ABB RAPID module: Module1.mod

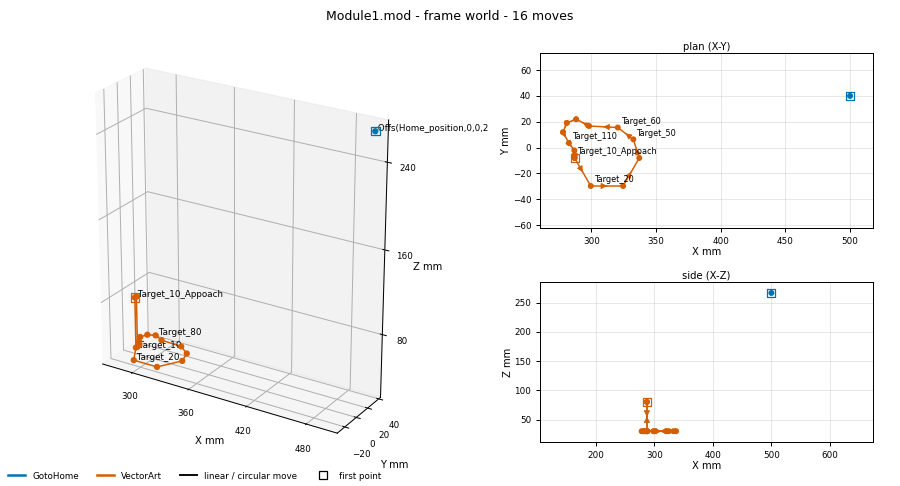
[picture p0: tool path of Module1.mod in frame world, 16 of 848 moves have a stored position in this frame; points joined in program order, loops and branches not executed]
MODULE Module1
    ! Define Global Constants
	CONST robtarget Home_position:=[[297,210,180],[0,0,1,0],[0,0,0,0],[9E+09,9E+09,9E+09,9E+09,9E+09,9E+09]];
	CONST robtarget Bottom_Left:=[[0,420,0],[0,0,1,0],[0,0,0,0],[9E+09,9E+09,9E+09,9E+09,9E+09,9E+09]];
	CONST robtarget Top_Left:=[[297,420,0],[0,0,1,0],[0,0,0,0],[9E+09,9E+09,9E+09,9E+09,9E+09,9E+09]];
	CONST robtarget Top_Right:=[[297,0,0],[0,0,1,0],[0,0,0,0],[9E+09,9E+09,9E+09,9E+09,9E+09,9E+09]];
	CONST robtarget Bottom_Right:=[[0,0,0],[0,0,1,0],[0,0,0,0],[9E+09,9E+09,9E+09,9E+09,9E+09,9E+09]];
	CONST robtarget Target_10_Appoach:=[[84,162,13.48],[0,-0.707106781,0.707106781,0],[-1,0,-2,0],[9E+09,9E+09,9E+09,9E+09,9E+09,9E+09]];
	CONST robtarget Target_10:=[[84,162,-36.52],[0,-0.707106781,0.707106781,0],[-1,0,-2,0],[9E+09,9E+09,9E+09,9E+09,9E+09,9E+09]];
	CONST robtarget Target_20:=[[96.5,140.349364905,-36.52],[0,-0.707106781,0.707106781,0],[-1,0,-2,0],[9E+09,9E+09,9E+09,9E+09,9E+09,9E+09]];
	CONST robtarget Target_30:=[[121.5,140.349364905,-36.52],[0,-0.707106781,0.707106781,0],[-1,0,-2,0],[9E+09,9E+09,9E+09,9E+09,9E+09,9E+09]];
	CONST robtarget Target_40:=[[134,162,-36.52],[0,-0.707106781,0.707106781,0],[-1,0,-2,0],[9E+09,9E+09,9E+09,9E+09,9E+09,9E+09]];
	CONST robtarget Target_50:=[[129.425575437,176.415126364,-36.52],[0,-0.707106781,0.707106781,0],[0,0,-1,0],[9E+09,9E+09,9E+09,9E+09,9E+09,9E+09]];
	CONST robtarget Target_60:=[[117.376330553,185.554980078,-36.52],[0,-0.707106781,0.707106781,0],[0,0,-1,0],[9E+09,9E+09,9E+09,9E+09,9E+09,9E+09]];
	CONST robtarget Target_70:=[[95.190280659,186.713087817,-36.52],[0,-0.707106781,0.707106781,0],[0,0,-1,0],[9E+09,9E+09,9E+09,9E+09,9E+09,9E+09]];
	CONST robtarget Target_80:=[[85.203125494,191.997936789,-36.52],[0,-0.707106781,0.707106781,0],[0,0,-1,0],[9E+09,9E+09,9E+09,9E+09,9E+09,9E+09]];
	CONST robtarget Target_90:=[[78.001116337,189.142522487,-36.52],[0,-0.707106781,0.707106781,0],[0,0,-1,0],[9E+09,9E+09,9E+09,9E+09,9E+09,9E+09]];
	CONST robtarget Target_100:=[[75,182,-36.52],[0,-0.707106781,0.707106781,0],[0,0,-1,0],[9E+09,9E+09,9E+09,9E+09,9E+09,9E+09]];
	CONST robtarget Target_110:=[[79.573343373,173.600512048,-36.52],[0,-0.707106781,0.707106781,0],[0,0,-1,0],[9E+09,9E+09,9E+09,9E+09,9E+09,9E+09]];
	CONST robtarget Target_120:=[[83.780815333,167.881241697,-36.52],[0,-0.707106781,0.707106781,0],[-1,0,-2,0],[9E+09,9E+09,9E+09,9E+09,9E+09,9E+09]];
	CONST robtarget Target_130:=[[84.104776248,164.286445783,-36.52],[0,-0.707106781,0.707106781,0],[-1,0,-2,0],[9E+09,9E+09,9E+09,9E+09,9E+09,9E+09]];
	CONST robtarget Target_130_Depart:=[[84.104776248,164.286445783,13.48],[0,-0.707106781,0.707106781,0],[-1,0,-2,0],[9E+09,9E+09,9E+09,9E+09,9E+09,9E+09]];

    !***********************************************************
    !
    ! Module:  Module1
    !
    ! Disclaimer:
    !    This module was written as part of my submission for Middlesex University's
    !    2017-2018 Mobile Robots and Manipulators module.
    !
    !    Note that this script in intended for GOOD and not for EVIL.
    !    Please do not use in any negative context, at least not without prior consent from
    !    the author of this script.
    !
    ! Author:
    !    Chibuike Okpaluba <co607@live.mdx.ac.uk> M00543047
    !
    ! Module Tutor:
    !    Dr Aleksander Zivanovic <a.zivanovic@mdx.ac.uk>
    !
    ! Description:
    !   This module contains all the necessary procedures and functions required to
    !
    !   1. Draw manually defined characters on a given worksurface using a preselected tool.
    !   2. Draw selected artworks on a given worksurface using a preselected tool.
    !   3. Draw the vector artwork on a given worksurface using a preselected tool.
    !   4. Automatically generate artworks for users that select the special option.
    !
    !   -- THE ENTRY POINT FOR THIS MODULE IS MAIN --
    !
    ! Version:
    !   v1.0
    !
    ! Questions and Answers:
    !   For more information please email the author of the module
    !
    !
    ! Thank you.
    !
    !***********************************************************


    !***********************************************************
    !
    ! Procedure main
    !   This the entry point of this module.
    !
    !   This procedure executes other procedures based on user inputs
    !***********************************************************
    PROC Main()
        ! Define Function Variables
        VAR num font_size := 0.5;
        VAR string answer := "Blink";

        ! GO Home and Wait 10 seconds
        GotoHome;
        !WaitTime 10;

        ! Get Data from the user
        TPReadFK reg1, "Select Drawing?", "Initials", "Artwork", "Vector", "Your String", "Special";

        ! Execute based on user data
        IF reg1 = 1 THEN
            TPWrite "Drawing initials: ''C.O''";
            DrawIntials font_size;

        ELSEIF reg1 = 2 THEN
            TPWrite "Drawing Artwork";
            DrawArtwork v100, v50, 100, 25, -10, 50;

        ELSEIF reg1 = 3 THEN
            TPWrite "Drawing Vector Art";
            VectorArt;

        ELSEIF reg1 = 4 THEN
            ! Get Text from the user
            answer := UIAlphaEntry(\Header:="Blink UI",
                \Message:="Enter your text?"
                \Icon:=iconInfo
                \InitString:="Your Text");

            ! Get font size from the user
            TPReadNum reg1, "Enter your font_size";

            ! Draw the users string
            DrawString answer, reg1, v80, v50, 10, 10, -10, 50;

        ELSEIF reg1 = 5 THEN
            ! Start special art
            MakeArtwork;

        ELSE
            TPWrite "Invalid selection";

        ENDIF

    ENDPROC

    !***********************************************************
    !
    ! Procedure GotoHome
    !   This Procedure moves the arm to the GLOBAL defined home position
    !
    ! Example
    !   GotoHome
    !
    !***********************************************************
    PROC GotoHome()
        ! Move arm joints to home position
        MoveJ Offs(Home_position, 0, 0, 20),v1000,z100,tool0\WObj:=WorkSurface;
    ENDPROC

    !***********************************************************
    !
    ! Procedure DrawIntials
    !   This procedure draws the intials on the work surface
    !
    ! Example
    !   VAR num font_size := 1.0;
    !   DrawIntials font_size;
    !
    !***********************************************************
    PROC DrawIntials(num font_size)
        DrawString "#Chib!", font_size, v100, v50, 5, 5, -10, 50;
        DrawString "#Chib!", font_size, v100, v50, 5, 65, -10, 50;
        DrawString "#Chib!", font_size, v100, v50, 5, 125, -10, 50;
        DrawString "#Chib!", font_size, v100, v50, 5, 185, -10, 50;
    ENDPROC

    !***********************************************************
    !
    ! Procedure MakeArtwork
    !   This procedure creates an artwork for the user based on the users string input
    !
    ! Example
    !   MakeArtwork;
    !
    !***********************************************************
    PROC MakeArtwork()
        VAR num page_width := 290;
        VAR num x_padding := 55;
        VAR num y_padding := 50;
        VAR string input_string := "";
        VAR num font_size := 0;

        VAR num z_offset := -10;
        VAR num penup_offset := 50;

        VAR num art_option;

        ! Get User's text
        input_string := UIAlphaEntry(\Header:="Blink UI",
                \Message:="Enter your text?"
                \Icon:=iconInfo
                \InitString:="#YourText");

        ! Drawing border art
        DrawArtWork_ArtBorder 0.45, v100, v50, 0, 0, z_offset, penup_offset;

        ! Calculate ideal font size
        font_size := get_ideal_font_size(input_string, page_width, x_padding);

        y_padding := 200 - (font_size * 50);
        DrawString input_string, font_size, v100, v50, x_padding, y_padding, z_offset, penup_offset;

        ! Get art option from the user
        TPReadFK reg1, "Select Art Option?", "House", stEmpty, stEmpty, stEmpty, "Glasses";
        art_option := reg1;

        IF art_option = 5 THEN
            y_padding := y_padding + (50 * font_size) + 5;
            x_padding := 96;
            DrawArtWork_Glasses 0.47, v100, v50, x_padding, y_padding, z_offset, penup_offset;
        ELSEIF art_option = 1 THEN
            y_padding := y_padding + (50 * font_size) + 5;
            x_padding := 106;
            DrawArtWork_House 0.38, v100, v50, x_padding, y_padding, z_offset, penup_offset;
        ENDIF
    ENDPROC

    !***********************************************************
    !
    ! Procedure DrawArtwork
    !   This procedure draws my artwork on the work surface
    !
    ! Example
    !   VAR speeddata approach_speed := v100;  // Approach speed for arm
    !   VAR speeddata write_speed := v80;      // Write speed for arm
    !   VAR num x_offset := 0;                 // x offset from worksurface origin
    !   VAR num y_offset := 0;                 // y offset from worksurface origin
    !   VAR num z_offset := 0;                 // z offset from worksurface origin
    !   VAR num pen_offset := 30;              // Defines pen position for pen up
    !
    !   DrawArtwork approach_speed, write_speed, x_offset, y_offset, z_offset, penup_offset;
    !
    !***********************************************************
    PROC DrawArtwork(speeddata approach_speed, speeddata write_speed, num x_offset, num y_offset, num z_offset, num penup_offset)
        ! Define all points for artwork
        VAR pos pos0{17} := [[153.29999999999998, 151.89999999999998, 0],[152.6, 152.6, 0],[152.6, 154.0, 0],[153.29999999999998, 154.7, 0],[153.29999999999998, 155.39999999999998, 0],[155.39999999999998, 157.5, 0],[158.2, 157.5, 0],[160.29999999999998, 155.39999999999998, 0],[160.29999999999998, 154.7, 0],[161.0, 154.0, 0],[161.0, 152.6, 0],[160.29999999999998, 151.89999999999998, 0],[160.29999999999998, 151.2, 0],[158.89999999999998, 149.79999999999998, 0],[154.7, 149.79999999999998, 0],[153.29999999999998, 151.2, 0],[153.29999999999998, 151.89999999999998, 0]];
        VAR pos pos1{10} := [[154.7, 152.6, 0],[155.39999999999998, 151.89999999999998, 0],[156.79999999999998, 151.89999999999998, 0],[157.5, 152.6, 0],[157.5, 154.0, 0],[156.79999999999998, 154.0, 0],[156.1, 154.7, 0],[155.39999999999998, 154.0, 0],[154.7, 154.0, 0],[154.7, 152.6, 0]];
        VAR pos pos2{17} := [[153.29999999999998, 109.19999999999999, 0],[152.6, 109.89999999999999, 0],[152.6, 111.3, 0],[153.29999999999998, 112.0, 0],[153.29999999999998, 112.69999999999999, 0],[155.39999999999998, 114.8, 0],[158.2, 114.8, 0],[160.29999999999998, 112.69999999999999, 0],[160.29999999999998, 112.0, 0],[161.0, 111.3, 0],[161.0, 109.89999999999999, 0],[160.29999999999998, 109.19999999999999, 0],[160.29999999999998, 108.5, 0],[158.89999999999998, 107.1, 0],[154.7, 107.1, 0],[153.29999999999998, 108.5, 0],[153.29999999999998, 109.19999999999999, 0]];
        VAR pos pos3{10} := [[154.7, 109.89999999999999, 0],[155.39999999999998, 109.19999999999999, 0],[156.79999999999998, 109.19999999999999, 0],[157.5, 109.89999999999999, 0],[157.5, 111.3, 0],[156.79999999999998, 111.3, 0],[156.1, 112.0, 0],[155.39999999999998, 111.3, 0],[154.7, 111.3, 0],[154.7, 109.89999999999999, 0]];
        VAR pos pos4{19} := [[153.29999999999998, 82.6, 0],[152.6, 83.3, 0],[152.6, 84.69999999999999, 0],[153.29999999999998, 85.39999999999999, 0],[153.29999999999998, 86.1, 0],[155.39999999999998, 88.19999999999999, 0],[158.2, 88.19999999999999, 0],[160.29999999999998, 86.1, 0],[160.29999999999998, 85.39999999999999, 0],[161.0, 84.69999999999999, 0],[161.0, 83.3, 0],[160.29999999999998, 82.6, 0],[160.29999999999998, 81.89999999999999, 0],[159.6, 81.19999999999999, 0],[158.89999999999998, 81.19999999999999, 0],[158.2, 80.5, 0],[154.7, 80.5, 0],[153.29999999999998, 81.89999999999999, 0],[153.29999999999998, 82.6, 0]];
        VAR pos pos5{10} := [[154.7, 83.3, 0],[155.39999999999998, 82.6, 0],[156.79999999999998, 82.6, 0],[157.5, 83.3, 0],[157.5, 84.69999999999999, 0],[156.79999999999998, 84.69999999999999, 0],[156.1, 85.39999999999999, 0],[155.39999999999998, 84.69999999999999, 0],[154.7, 84.69999999999999, 0],[154.7, 83.3, 0]];
        VAR pos pos6{57} := [[126.69999999999999, 172.89999999999998, 0],[125.99999999999999, 173.6, 0],[125.99999999999999, 177.79999999999998, 0],[126.69999999999999, 178.5, 0],[126.69999999999999, 180.6, 0],[127.39999999999999, 181.29999999999998, 0],[127.39999999999999, 182.0, 0],[132.29999999999998, 186.89999999999998, 0],[133.0, 186.89999999999998, 0],[134.39999999999998, 188.29999999999998, 0],[135.79999999999998, 188.29999999999998, 0],[136.5, 189.0, 0],[137.2, 189.0, 0],[137.89999999999998, 189.7, 0],[147.7, 189.7, 0],[148.39999999999998, 189.0, 0],[149.79999999999998, 189.0, 0],[150.5, 188.29999999999998, 0],[151.2, 188.29999999999998, 0],[151.89999999999998, 187.6, 0],[152.6, 187.6, 0],[153.29999999999998, 186.89999999999998, 0],[154.0, 186.89999999999998, 0],[158.89999999999998, 182.0, 0],[158.89999999999998, 181.29999999999998, 0],[159.6, 180.6, 0],[159.6, 178.5, 0],[160.29999999999998, 177.79999999999998, 0],[160.29999999999998, 173.6, 0],[159.6, 172.89999999999998, 0],[159.6, 171.5, 0],[158.89999999999998, 170.79999999999998, 0],[158.89999999999998, 170.1, 0],[158.2, 169.39999999999998, 0],[158.2, 168.7, 0],[154.7, 165.2, 0],[154.0, 165.2, 0],[152.6, 163.79999999999998, 0],[151.89999999999998, 163.79999999999998, 0],[151.2, 163.1, 0],[149.79999999999998, 163.1, 0],[149.1, 162.39999999999998, 0],[147.0, 162.39999999999998, 0],[146.29999999999998, 161.7, 0],[139.29999999999998, 161.7, 0],[138.6, 162.39999999999998, 0],[136.5, 162.39999999999998, 0],[135.79999999999998, 163.1, 0],[135.1, 163.1, 0],[134.39999999999998, 163.79999999999998, 0],[133.7, 163.79999999999998, 0],[133.0, 164.5, 0],[132.29999999999998, 164.5, 0],[127.39999999999999, 169.39999999999998, 0],[127.39999999999999, 170.1, 0],[126.69999999999999, 170.79999999999998, 0],[126.69999999999999, 172.89999999999998, 0]];
        VAR pos pos7{96} := [[133.7, 176.39999999999998, 0],[135.1, 176.39999999999998, 0],[135.79999999999998, 177.1, 0],[137.89999999999998, 177.1, 0],[138.6, 176.39999999999998, 0],[138.6, 175.7, 0],[137.89999999999998, 175.0, 0],[137.2, 175.0, 0],[136.5, 174.29999999999998, 0],[135.1, 174.29999999999998, 0],[134.39999999999998, 173.6, 0],[134.39999999999998, 172.89999999999998, 0],[135.79999999999998, 171.5, 0],[135.79999999999998, 170.79999999999998, 0],[136.5, 170.1, 0],[137.2, 170.1, 0],[137.89999999999998, 169.39999999999998, 0],[138.6, 169.39999999999998, 0],[141.39999999999998, 172.2, 0],[142.1, 172.2, 0],[143.5, 170.79999999999998, 0],[140.7, 168.0, 0],[141.39999999999998, 168.0, 0],[142.1, 167.29999999999998, 0],[146.29999999999998, 167.29999999999998, 0],[146.29999999999998, 170.1, 0],[147.0, 170.79999999999998, 0],[147.7, 170.79999999999998, 0],[148.39999999999998, 170.1, 0],[148.39999999999998, 167.29999999999998, 0],[149.79999999999998, 167.29999999999998, 0],[150.5, 168.0, 0],[151.89999999999998, 168.0, 0],[151.89999999999998, 168.7, 0],[149.79999999999998, 170.79999999999998, 0],[149.79999999999998, 171.5, 0],[150.5, 172.2, 0],[151.2, 172.2, 0],[154.0, 169.39999999999998, 0],[156.1, 171.5, 0],[156.1, 172.2, 0],[156.79999999999998, 172.89999999999998, 0],[156.1, 172.89999999999998, 0],[155.39999999999998, 173.6, 0],[153.29999999999998, 173.6, 0],[152.6, 174.29999999999998, 0],[154.0, 175.7, 0],[157.5, 175.7, 0],[157.5, 176.39999999999998, 0],[156.79999999999998, 177.1, 0],[156.79999999999998, 178.5, 0],[156.1, 179.2, 0],[156.1, 179.89999999999998, 0],[155.39999999999998, 179.89999999999998, 0],[154.7, 179.2, 0],[154.0, 179.2, 0],[153.29999999999998, 178.5, 0],[152.6, 178.5, 0],[151.89999999999998, 177.79999999999998, 0],[151.2, 177.79999999999998, 0],[149.79999999999998, 179.2, 0],[151.2, 180.6, 0],[151.89999999999998, 180.6, 0],[152.6, 181.29999999999998, 0],[153.29999999999998, 181.29999999999998, 0],[154.0, 182.0, 0],[153.29999999999998, 182.0, 0],[151.89999999999998, 183.39999999999998, 0],[150.5, 183.39999999999998, 0],[147.7, 180.6, 0],[146.29999999999998, 182.0, 0],[147.7, 183.39999999999998, 0],[147.7, 184.79999999999998, 0],[143.5, 184.79999999999998, 0],[143.5, 182.0, 0],[142.79999999999998, 181.29999999999998, 0],[141.39999999999998, 182.7, 0],[141.39999999999998, 184.79999999999998, 0],[140.7, 184.1, 0],[139.29999999999998, 184.1, 0],[138.6, 183.39999999999998, 0],[137.89999999999998, 183.39999999999998, 0],[137.89999999999998, 182.7, 0],[140.0, 180.6, 0],[140.0, 179.89999999999998, 0],[139.29999999999998, 179.2, 0],[138.6, 179.2, 0],[137.89999999999998, 179.89999999999998, 0],[137.2, 179.89999999999998, 0],[135.79999999999998, 181.29999999999998, 0],[135.1, 181.29999999999998, 0],[135.1, 180.6, 0],[134.39999999999998, 179.89999999999998, 0],[134.39999999999998, 179.2, 0],[133.7, 178.5, 0],[133.7, 176.39999999999998, 0]];
        VAR pos pos8{35} := [[125.99999999999999, 96.6, 0],[125.99999999999999, 97.3, 0],[126.69999999999999, 98.0, 0],[126.69999999999999, 102.89999999999999, 0],[128.1, 104.3, 0],[129.5, 104.3, 0],[130.2, 103.6, 0],[132.29999999999998, 103.6, 0],[133.0, 102.89999999999999, 0],[135.1, 102.89999999999999, 0],[135.79999999999998, 102.19999999999999, 0],[137.89999999999998, 102.19999999999999, 0],[138.6, 101.5, 0],[141.39999999999998, 101.5, 0],[142.1, 100.8, 0],[144.89999999999998, 100.8, 0],[145.6, 100.1, 0],[149.79999999999998, 100.1, 0],[150.5, 99.39999999999999, 0],[158.89999999999998, 99.39999999999999, 0],[159.6, 98.69999999999999, 0],[159.6, 96.6, 0],[160.29999999999998, 95.89999999999999, 0],[160.29999999999998, 94.5, 0],[159.6, 93.8, 0],[154.0, 93.8, 0],[153.29999999999998, 93.1, 0],[149.1, 93.1, 0],[148.39999999999998, 93.8, 0],[137.89999999999998, 93.8, 0],[137.2, 94.5, 0],[132.29999999999998, 94.5, 0],[131.6, 95.19999999999999, 0],[127.39999999999999, 95.19999999999999, 0],[125.99999999999999, 96.6, 0]];
        VAR pos pos9{23} := [[132.29999999999998, 100.1, 0],[133.0, 99.39999999999999, 0],[133.7, 99.39999999999999, 0],[134.39999999999998, 98.69999999999999, 0],[135.1, 98.69999999999999, 0],[135.79999999999998, 98.0, 0],[137.2, 98.0, 0],[137.89999999999998, 97.3, 0],[139.29999999999998, 97.3, 0],[140.0, 96.6, 0],[142.1, 96.6, 0],[142.79999999999998, 97.3, 0],[141.39999999999998, 97.3, 0],[140.7, 98.0, 0],[138.6, 98.0, 0],[137.89999999999998, 98.69999999999999, 0],[136.5, 98.69999999999999, 0],[135.79999999999998, 99.39999999999999, 0],[135.1, 99.39999999999999, 0],[134.39999999999998, 100.1, 0],[133.0, 100.1, 0],[132.29999999999998, 100.8, 0],[132.29999999999998, 100.1, 0]];
        VAR pos pos10{23} := [[125.99999999999999, 40.599999999999994, 0],[127.39999999999999, 42.0, 0],[128.1, 42.0, 0],[129.5, 40.599999999999994, 0],[130.9, 40.599999999999994, 0],[130.9, 41.3, 0],[133.0, 43.4, 0],[134.39999999999998, 43.4, 0],[135.1, 42.699999999999996, 0],[135.79999999999998, 42.699999999999996, 0],[136.5, 42.0, 0],[136.5, 41.3, 0],[137.2, 40.599999999999994, 0],[137.2, 39.199999999999996, 0],[136.5, 38.5, 0],[136.5, 37.8, 0],[135.1, 36.4, 0],[131.6, 36.4, 0],[130.9, 37.099999999999994, 0],[130.2, 37.099999999999994, 0],[128.79999999999998, 38.5, 0],[128.1, 38.5, 0],[125.99999999999999, 40.599999999999994, 0]];
        VAR pos pos11{9} := [[132.29999999999998, 39.9, 0],[133.0, 39.199999999999996, 0],[134.39999999999998, 39.199999999999996, 0],[135.1, 39.9, 0],[135.1, 40.599999999999994, 0],[134.39999999999998, 41.3, 0],[133.0, 41.3, 0],[132.29999999999998, 40.599999999999994, 0],[132.29999999999998, 39.9, 0]];
        VAR pos pos12{42} := [[125.99999999999999, 205.79999999999998, 0],[125.3, 206.5, 0],[125.3, 207.2, 0],[125.99999999999999, 207.89999999999998, 0],[125.99999999999999, 208.6, 0],[126.69999999999999, 209.29999999999998, 0],[126.69999999999999, 211.39999999999998, 0],[127.39999999999999, 212.1, 0],[128.79999999999998, 210.7, 0],[130.2, 210.7, 0],[130.2, 211.39999999999998, 0],[130.9, 212.1, 0],[131.6, 212.1, 0],[132.29999999999998, 211.39999999999998, 0],[132.29999999999998, 210.0, 0],[133.0, 210.0, 0],[133.7, 209.29999999999998, 0],[135.1, 209.29999999999998, 0],[135.79999999999998, 210.0, 0],[137.2, 208.6, 0],[136.5, 207.89999999999998, 0],[136.5, 207.2, 0],[137.2, 206.5, 0],[135.79999999999998, 205.1, 0],[134.39999999999998, 206.5, 0],[133.7, 206.5, 0],[133.0, 207.2, 0],[132.29999999999998, 207.2, 0],[132.29999999999998, 206.5, 0],[131.6, 205.79999999999998, 0],[133.0, 204.39999999999998, 0],[132.29999999999998, 203.7, 0],[131.6, 203.7, 0],[130.9, 204.39999999999998, 0],[129.5, 204.39999999999998, 0],[128.1, 203.0, 0],[127.39999999999999, 203.0, 0],[126.69999999999999, 203.7, 0],[127.39999999999999, 204.39999999999998, 0],[127.39999999999999, 205.1, 0],[126.69999999999999, 205.79999999999998, 0],[125.99999999999999, 205.79999999999998, 0]];
        VAR pos pos13{22} := [[125.3, 197.39999999999998, 0],[125.3, 199.5, 0],[125.99999999999999, 200.2, 0],[125.99999999999999, 200.89999999999998, 0],[126.69999999999999, 201.6, 0],[127.39999999999999, 201.6, 0],[128.1, 202.29999999999998, 0],[130.2, 202.29999999999998, 0],[130.9, 201.6, 0],[131.6, 201.6, 0],[132.29999999999998, 200.89999999999998, 0],[133.0, 200.89999999999998, 0],[136.5, 197.39999999999998, 0],[135.1, 196.0, 0],[134.39999999999998, 196.7, 0],[133.7, 196.7, 0],[132.29999999999998, 198.1, 0],[131.6, 198.1, 0],[131.6, 196.7, 0],[130.2, 195.29999999999998, 0],[127.39999999999999, 195.29999999999998, 0],[125.3, 197.39999999999998, 0]];
        VAR pos pos14{9} := [[127.39999999999999, 198.1, 0],[128.1, 197.39999999999998, 0],[129.5, 197.39999999999998, 0],[130.2, 198.1, 0],[130.2, 198.79999999999998, 0],[129.5, 199.5, 0],[128.1, 199.5, 0],[127.39999999999999, 198.79999999999998, 0],[127.39999999999999, 198.1, 0]];
        VAR pos pos15{55} := [[125.99999999999999, 128.1, 0],[125.3, 128.79999999999998, 0],[125.3, 135.79999999999998, 0],[125.99999999999999, 136.5, 0],[125.99999999999999, 138.6, 0],[126.69999999999999, 139.29999999999998, 0],[126.69999999999999, 140.7, 0],[130.9, 144.89999999999998, 0],[132.29999999999998, 144.89999999999998, 0],[133.0, 145.6, 0],[138.6, 145.6, 0],[139.29999999999998, 144.89999999999998, 0],[140.0, 144.89999999999998, 0],[140.7, 144.2, 0],[141.39999999999998, 144.2, 0],[144.89999999999998, 140.7, 0],[144.89999999999998, 139.29999999999998, 0],[145.6, 138.6, 0],[145.6, 135.1, 0],[144.89999999999998, 134.39999999999998, 0],[144.89999999999998, 133.0, 0],[142.1, 130.2, 0],[141.39999999999998, 130.2, 0],[146.29999999999998, 130.2, 0],[147.0, 129.5, 0],[156.79999999999998, 129.5, 0],[157.5, 128.79999999999998, 0],[160.29999999999998, 128.79999999999998, 0],[161.0, 128.1, 0],[161.0, 125.99999999999999, 0],[161.7, 125.3, 0],[161.0, 124.6, 0],[160.29999999999998, 124.6, 0],[159.6, 123.89999999999999, 0],[144.2, 123.89999999999999, 0],[144.2, 121.1, 0],[143.5, 120.39999999999999, 0],[141.39999999999998, 120.39999999999999, 0],[140.7, 121.1, 0],[140.7, 121.8, 0],[140.0, 122.49999999999999, 0],[140.0, 123.89999999999999, 0],[137.2, 123.89999999999999, 0],[137.2, 121.1, 0],[136.5, 120.39999999999999, 0],[133.7, 120.39999999999999, 0],[133.0, 121.1, 0],[133.0, 123.89999999999999, 0],[132.29999999999998, 123.19999999999999, 0],[130.2, 123.19999999999999, 0],[130.2, 120.39999999999999, 0],[129.5, 119.69999999999999, 0],[126.69999999999999, 119.69999999999999, 0],[125.99999999999999, 120.39999999999999, 0],[125.99999999999999, 128.1, 0]];
        VAR pos pos16{42} := [[129.5, 130.9, 0],[134.39999999999998, 130.9, 0],[133.7, 130.9, 0],[132.29999999999998, 132.29999999999998, 0],[132.29999999999998, 133.7, 0],[131.6, 134.39999999999998, 0],[131.6, 136.5, 0],[132.29999999999998, 137.2, 0],[132.29999999999998, 137.89999999999998, 0],[133.7, 139.29999999999998, 0],[134.39999999999998, 139.29999999999998, 0],[135.1, 140.0, 0],[137.2, 140.0, 0],[139.29999999999998, 137.89999999999998, 0],[139.29999999999998, 135.79999999999998, 0],[137.89999999999998, 134.39999999999998, 0],[137.2, 135.1, 0],[137.2, 136.5, 0],[135.79999999999998, 136.5, 0],[135.79999999999998, 134.39999999999998, 0],[136.5, 133.7, 0],[137.2, 133.7, 0],[137.89999999999998, 133.0, 0],[139.29999999999998, 133.0, 0],[140.0, 133.7, 0],[140.7, 133.7, 0],[142.1, 135.1, 0],[142.1, 137.89999999999998, 0],[141.39999999999998, 138.6, 0],[141.39999999999998, 139.29999999999998, 0],[140.7, 140.0, 0],[140.0, 140.0, 0],[139.29999999999998, 140.7, 0],[133.7, 140.7, 0],[133.0, 140.0, 0],[132.29999999999998, 140.0, 0],[130.9, 138.6, 0],[130.9, 137.89999999999998, 0],[130.2, 137.2, 0],[130.2, 136.5, 0],[129.5, 135.79999999999998, 0],[129.5, 130.9, 0]];
        VAR pos pos17{41} := [[125.99999999999999, 28.7, 0],[125.3, 29.4, 0],[125.99999999999999, 30.099999999999998, 0],[125.99999999999999, 30.799999999999997, 0],[125.3, 31.499999999999996, 0],[126.69999999999999, 32.9, 0],[127.39999999999999, 32.199999999999996, 0],[128.1, 32.199999999999996, 0],[128.79999999999998, 31.499999999999996, 0],[130.2, 31.499999999999996, 0],[130.2, 32.9, 0],[129.5, 33.599999999999994, 0],[130.9, 35.0, 0],[131.6, 34.3, 0],[133.7, 34.3, 0],[133.7, 35.0, 0],[134.39999999999998, 35.699999999999996, 0],[135.79999999999998, 34.3, 0],[135.1, 33.599999999999994, 0],[135.79999999999998, 32.9, 0],[135.79999999999998, 32.199999999999996, 0],[136.5, 32.199999999999996, 0],[137.2, 31.499999999999996, 0],[137.2, 30.799999999999997, 0],[135.79999999999998, 29.4, 0],[135.79999999999998, 27.299999999999997, 0],[135.1, 26.599999999999998, 0],[134.39999999999998, 26.599999999999998, 0],[133.7, 27.299999999999997, 0],[133.7, 28.0, 0],[132.29999999999998, 28.0, 0],[132.29999999999998, 27.299999999999997, 0],[131.6, 26.599999999999998, 0],[130.9, 26.599999999999998, 0],[130.2, 27.299999999999997, 0],[130.2, 28.0, 0],[129.5, 28.7, 0],[128.79999999999998, 28.7, 0],[128.1, 29.4, 0],[127.39999999999999, 28.7, 0],[125.99999999999999, 28.7, 0]];
        VAR pos pos18{137} := [[125.3, 59.49999999999999, 0],[124.6, 60.199999999999996, 0],[124.6, 61.599999999999994, 0],[125.3, 62.3, 0],[125.99999999999999, 62.3, 0],[125.99999999999999, 67.19999999999999, 0],[125.3, 67.19999999999999, 0],[124.6, 67.89999999999999, 0],[124.6, 69.3, 0],[125.3, 70.0, 0],[125.99999999999999, 69.3, 0],[127.39999999999999, 69.3, 0],[129.5, 71.39999999999999, 0],[129.5, 72.8, 0],[128.79999999999998, 73.5, 0],[129.5, 74.19999999999999, 0],[130.9, 74.19999999999999, 0],[132.29999999999998, 72.8, 0],[133.0, 72.8, 0],[133.7, 73.5, 0],[134.39999999999998, 73.5, 0],[135.1, 72.8, 0],[135.1, 71.39999999999999, 0],[131.6, 67.89999999999999, 0],[131.6, 67.19999999999999, 0],[130.9, 66.5, 0],[130.9, 61.599999999999994, 0],[131.6, 60.9, 0],[131.6, 60.199999999999996, 0],[133.0, 58.8, 0],[133.0, 58.099999999999994, 0],[133.7, 57.4, 0],[134.39999999999998, 57.4, 0],[135.79999999999998, 56.0, 0],[137.2, 56.0, 0],[137.89999999999998, 55.3, 0],[144.2, 55.3, 0],[144.89999999999998, 56.0, 0],[146.29999999999998, 56.0, 0],[149.79999999999998, 59.49999999999999, 0],[149.79999999999998, 60.199999999999996, 0],[150.5, 60.9, 0],[150.5, 62.3, 0],[151.2, 62.99999999999999, 0],[151.2, 65.1, 0],[150.5, 65.8, 0],[150.5, 67.19999999999999, 0],[147.7, 70.0, 0],[145.6, 70.0, 0],[144.2, 71.39999999999999, 0],[144.2, 72.8, 0],[144.89999999999998, 73.5, 0],[146.29999999999998, 73.5, 0],[147.0, 74.19999999999999, 0],[147.0, 74.89999999999999, 0],[147.7, 75.6, 0],[148.39999999999998, 74.89999999999999, 0],[148.39999999999998, 74.19999999999999, 0],[149.1, 73.5, 0],[151.89999999999998, 73.5, 0],[151.89999999999998, 74.19999999999999, 0],[152.6, 74.89999999999999, 0],[153.29999999999998, 74.89999999999999, 0],[154.0, 74.19999999999999, 0],[154.0, 72.1, 0],[156.79999999999998, 69.3, 0],[157.5, 70.0, 0],[158.89999999999998, 70.0, 0],[159.6, 69.3, 0],[159.6, 68.6, 0],[158.2, 67.19999999999999, 0],[157.5, 67.19999999999999, 0],[157.5, 66.5, 0],[158.2, 65.8, 0],[158.2, 62.3, 0],[160.29999999999998, 62.3, 0],[161.0, 61.599999999999994, 0],[161.0, 60.9, 0],[159.6, 59.49999999999999, 0],[158.89999999999998, 60.199999999999996, 0],[157.5, 60.199999999999996, 0],[157.5, 58.8, 0],[156.79999999999998, 58.099999999999994, 0],[156.79999999999998, 57.4, 0],[157.5, 57.4, 0],[158.89999999999998, 56.0, 0],[158.89999999999998, 55.3, 0],[158.2, 54.599999999999994, 0],[156.79999999999998, 54.599999999999994, 0],[156.1, 55.3, 0],[155.39999999999998, 55.3, 0],[152.6, 52.5, 0],[153.29999999999998, 51.8, 0],[153.29999999999998, 51.099999999999994, 0],[154.0, 50.4, 0],[152.6, 49.0, 0],[151.2, 50.4, 0],[151.2, 51.099999999999994, 0],[149.1, 51.099999999999994, 0],[148.39999999999998, 50.4, 0],[146.29999999999998, 50.4, 0],[145.6, 49.699999999999996, 0],[144.2, 49.699999999999996, 0],[144.2, 47.599999999999994, 0],[143.5, 46.9, 0],[142.79999999999998, 46.9, 0],[142.1, 47.599999999999994, 0],[142.1, 49.699999999999996, 0],[141.39999999999998, 49.699999999999996, 0],[140.7, 50.4, 0],[137.89999999999998, 50.4, 0],[137.2, 51.099999999999994, 0],[135.79999999999998, 51.099999999999994, 0],[135.1, 50.4, 0],[135.1, 49.699999999999996, 0],[134.39999999999998, 49.0, 0],[133.7, 49.0, 0],[132.29999999999998, 50.4, 0],[133.0, 51.099999999999994, 0],[133.0, 51.8, 0],[133.7, 52.5, 0],[133.0, 53.199999999999996, 0],[132.29999999999998, 53.199999999999996, 0],[130.9, 54.599999999999994, 0],[130.2, 53.9, 0],[129.5, 53.9, 0],[128.79999999999998, 53.199999999999996, 0],[128.1, 53.199999999999996, 0],[127.39999999999999, 53.9, 0],[127.39999999999999, 54.599999999999994, 0],[128.79999999999998, 56.0, 0],[128.79999999999998, 56.699999999999996, 0],[128.1, 57.4, 0],[128.1, 58.099999999999994, 0],[127.39999999999999, 58.8, 0],[127.39999999999999, 59.49999999999999, 0],[125.3, 59.49999999999999, 0]];
        VAR pos pos19{363} := [[0.7, 96.6, 0],[0.0, 97.3, 0],[0.0, 99.39999999999999, 0],[0.7, 100.1, 0],[1.4, 100.1, 0],[2.0999999999999996, 100.8, 0],[2.8, 100.8, 0],[3.5, 100.1, 0],[4.199999999999999, 100.1, 0],[4.8999999999999995, 100.8, 0],[0.7, 100.8, 0],[0.0, 101.5, 0],[0.0, 105.69999999999999, 0],[0.7, 106.39999999999999, 0],[4.199999999999999, 106.39999999999999, 0],[4.199999999999999, 107.1, 0],[0.7, 107.1, 0],[0.0, 107.8, 0],[0.0, 109.89999999999999, 0],[0.7, 110.6, 0],[4.8999999999999995, 110.6, 0],[4.8999999999999995, 111.3, 0],[0.7, 111.3, 0],[0.0, 112.0, 0],[0.0, 115.49999999999999, 0],[0.7, 116.19999999999999, 0],[1.4, 116.19999999999999, 0],[2.0999999999999996, 116.89999999999999, 0],[2.8, 116.19999999999999, 0],[3.5, 116.19999999999999, 0],[4.199999999999999, 116.89999999999999, 0],[4.8999999999999995, 116.89999999999999, 0],[0.7, 116.89999999999999, 0],[0.0, 117.6, 0],[0.0, 120.39999999999999, 0],[0.7, 121.1, 0],[4.8999999999999995, 121.1, 0],[4.199999999999999, 121.8, 0],[4.8999999999999995, 122.49999999999999, 0],[4.199999999999999, 123.19999999999999, 0],[3.5, 123.19999999999999, 0],[2.8, 122.49999999999999, 0],[2.0999999999999996, 122.49999999999999, 0],[1.4, 123.19999999999999, 0],[0.7, 123.19999999999999, 0],[0.0, 123.89999999999999, 0],[0.0, 124.6, 0],[0.7, 125.3, 0],[4.199999999999999, 125.3, 0],[4.8999999999999995, 125.99999999999999, 0],[4.8999999999999995, 126.69999999999999, 0],[4.199999999999999, 127.39999999999999, 0],[0.7, 127.39999999999999, 0],[0.0, 128.1, 0],[0.0, 130.2, 0],[0.7, 130.9, 0],[4.199999999999999, 130.9, 0],[4.199999999999999, 131.6, 0],[0.7, 131.6, 0],[0.0, 132.29999999999998, 0],[0.0, 134.39999999999998, 0],[0.7, 135.1, 0],[1.4, 135.1, 0],[2.0999999999999996, 135.79999999999998, 0],[2.8, 135.1, 0],[3.5, 135.1, 0],[4.8999999999999995, 136.5, 0],[4.8999999999999995, 137.2, 0],[4.199999999999999, 137.2, 0],[3.5, 137.89999999999998, 0],[2.8, 137.2, 0],[2.0999999999999996, 137.2, 0],[1.4, 137.89999999999998, 0],[0.7, 137.89999999999998, 0],[0.0, 138.6, 0],[0.0, 140.7, 0],[0.7, 141.39999999999998, 0],[16.099999999999998, 141.39999999999998, 0],[18.9, 144.2, 0],[18.9, 144.89999999999998, 0],[21.0, 147.0, 0],[44.8, 147.0, 0],[44.8, 147.7, 0],[44.099999999999994, 148.39999999999998, 0],[44.099999999999994, 149.1, 0],[44.8, 149.79999999999998, 0],[51.099999999999994, 149.79999999999998, 0],[51.099999999999994, 150.5, 0],[47.599999999999994, 150.5, 0],[46.9, 151.2, 0],[46.9, 154.0, 0],[47.599999999999994, 154.7, 0],[48.3, 154.0, 0],[49.0, 154.7, 0],[49.699999999999996, 154.0, 0],[51.099999999999994, 154.0, 0],[51.099999999999994, 156.1, 0],[49.699999999999996, 156.1, 0],[49.0, 156.79999999999998, 0],[48.3, 156.1, 0],[47.599999999999994, 156.1, 0],[46.9, 156.79999999999998, 0],[46.9, 158.2, 0],[47.599999999999994, 158.89999999999998, 0],[51.099999999999994, 158.89999999999998, 0],[51.099999999999994, 161.0, 0],[18.2, 161.0, 0],[17.5, 161.7, 0],[17.5, 163.79999999999998, 0],[18.2, 164.5, 0],[21.7, 164.5, 0],[21.7, 166.6, 0],[18.2, 166.6, 0],[17.5, 167.29999999999998, 0],[17.5, 170.79999999999998, 0],[18.9, 172.2, 0],[19.599999999999998, 172.2, 0],[20.299999999999997, 172.89999999999998, 0],[19.599999999999998, 173.6, 0],[18.9, 173.6, 0],[17.5, 175.0, 0],[17.5, 177.1, 0],[18.2, 177.79999999999998, 0],[21.7, 177.79999999999998, 0],[21.7, 178.5, 0],[22.4, 179.2, 0],[21.7, 179.89999999999998, 0],[18.2, 179.89999999999998, 0],[17.5, 180.6, 0],[17.5, 184.1, 0],[18.2, 184.79999999999998, 0],[51.099999999999994, 184.79999999999998, 0],[51.099999999999994, 185.5, 0],[47.599999999999994, 185.5, 0],[46.9, 186.2, 0],[46.9, 187.6, 0],[47.599999999999994, 188.29999999999998, 0],[50.4, 188.29999999999998, 0],[51.099999999999994, 187.6, 0],[51.099999999999994, 189.7, 0],[50.4, 189.7, 0],[49.699999999999996, 190.39999999999998, 0],[49.0, 190.39999999999998, 0],[48.3, 189.7, 0],[46.9, 191.1, 0],[46.9, 193.2, 0],[47.599999999999994, 193.89999999999998, 0],[51.099999999999994, 193.89999999999998, 0],[51.099999999999994, 194.6, 0],[18.2, 194.6, 0],[17.5, 195.29999999999998, 0],[17.5, 197.39999999999998, 0],[18.2, 198.1, 0],[22.4, 198.1, 0],[21.7, 198.79999999999998, 0],[21.7, 200.2, 0],[18.2, 200.2, 0],[17.5, 200.89999999999998, 0],[17.5, 204.39999999999998, 0],[18.9, 205.79999999999998, 0],[22.4, 205.79999999999998, 0],[21.7, 206.5, 0],[22.4, 207.2, 0],[21.7, 207.2, 0],[21.0, 207.89999999999998, 0],[18.2, 207.89999999999998, 0],[17.5, 208.6, 0],[17.5, 210.7, 0],[18.2, 211.39999999999998, 0],[21.7, 211.39999999999998, 0],[21.7, 212.1, 0],[22.4, 212.79999999999998, 0],[21.7, 213.5, 0],[18.2, 213.5, 0],[17.5, 214.2, 0],[17.5, 217.7, 0],[18.2, 218.39999999999998, 0],[51.099999999999994, 218.39999999999998, 0],[51.099999999999994, 219.1, 0],[47.599999999999994, 219.1, 0],[46.9, 219.79999999999998, 0],[46.9, 222.6, 0],[47.599999999999994, 223.29999999999998, 0],[48.3, 222.6, 0],[49.0, 223.29999999999998, 0],[49.699999999999996, 223.29999999999998, 0],[50.4, 222.6, 0],[51.099999999999994, 223.29999999999998, 0],[51.8, 222.6, 0],[52.5, 223.29999999999998, 0],[47.599999999999994, 223.29999999999998, 0],[46.9, 224.0, 0],[46.9, 228.2, 0],[47.599999999999994, 228.89999999999998, 0],[51.099999999999994, 228.89999999999998, 0],[51.099999999999994, 229.6, 0],[47.599999999999994, 229.6, 0],[46.9, 230.29999999999998, 0],[46.9, 232.39999999999998, 0],[47.599999999999994, 233.1, 0],[110.6, 233.1, 0],[111.3, 233.79999999999998, 0],[110.6, 234.49999999999997, 0],[111.3, 235.2, 0],[110.6, 235.89999999999998, 0],[110.6, 236.6, 0],[111.3, 237.29999999999998, 0],[116.89999999999999, 237.29999999999998, 0],[117.6, 236.6, 0],[117.6, 1.4, 0],[116.19999999999999, 0.0, 0],[114.1, 0.0, 0],[113.39999999999999, 0.7, 0],[111.3, 0.7, 0],[110.6, 1.4, 0],[110.6, 2.8, 0],[111.3, 3.5, 0],[110.6, 4.199999999999999, 0],[110.6, 4.8999999999999995, 0],[47.599999999999994, 4.8999999999999995, 0],[46.9, 5.6, 0],[46.9, 7.699999999999999, 0],[47.599999999999994, 8.399999999999999, 0],[51.099999999999994, 8.399999999999999, 0],[51.099999999999994, 10.5, 0],[47.599999999999994, 10.5, 0],[46.9, 11.2, 0],[46.9, 13.299999999999999, 0],[47.599999999999994, 14.0, 0],[48.3, 14.0, 0],[49.0, 14.7, 0],[50.4, 14.7, 0],[51.099999999999994, 14.0, 0],[51.099999999999994, 14.7, 0],[50.4, 15.399999999999999, 0],[49.699999999999996, 15.399999999999999, 0],[49.0, 14.7, 0],[48.3, 15.399999999999999, 0],[47.599999999999994, 15.399999999999999, 0],[46.9, 16.099999999999998, 0],[46.9, 18.2, 0],[47.599999999999994, 18.9, 0],[51.099999999999994, 18.9, 0],[51.099999999999994, 19.599999999999998, 0],[18.2, 19.599999999999998, 0],[17.5, 20.299999999999997, 0],[17.5, 23.799999999999997, 0],[18.2, 24.5, 0],[21.7, 24.5, 0],[21.7, 26.599999999999998, 0],[18.2, 26.599999999999998, 0],[17.5, 27.299999999999997, 0],[17.5, 29.4, 0],[18.9, 30.799999999999997, 0],[20.299999999999997, 30.799999999999997, 0],[21.0, 30.099999999999998, 0],[21.7, 30.099999999999998, 0],[21.7, 30.799999999999997, 0],[22.4, 31.499999999999996, 0],[21.0, 32.9, 0],[20.299999999999997, 32.199999999999996, 0],[19.599999999999998, 32.9, 0],[18.9, 32.199999999999996, 0],[17.5, 33.599999999999994, 0],[17.5, 37.099999999999994, 0],[18.2, 37.8, 0],[23.099999999999998, 37.8, 0],[23.099999999999998, 38.5, 0],[23.799999999999997, 39.199999999999996, 0],[23.099999999999998, 39.9, 0],[18.2, 39.9, 0],[17.5, 40.599999999999994, 0],[17.5, 42.699999999999996, 0],[18.2, 43.4, 0],[51.099999999999994, 43.4, 0],[51.099999999999994, 44.099999999999994, 0],[47.599999999999994, 44.099999999999994, 0],[46.9, 44.8, 0],[46.9, 46.9, 0],[48.3, 48.3, 0],[49.699999999999996, 48.3, 0],[50.4, 47.599999999999994, 0],[51.099999999999994, 47.599999999999994, 0],[51.8, 48.3, 0],[52.5, 48.3, 0],[52.5, 49.699999999999996, 0],[51.8, 50.4, 0],[51.099999999999994, 49.699999999999996, 0],[50.4, 50.4, 0],[48.3, 50.4, 0],[47.599999999999994, 49.699999999999996, 0],[46.9, 50.4, 0],[46.9, 51.8, 0],[47.599999999999994, 52.5, 0],[52.5, 52.5, 0],[52.5, 53.199999999999996, 0],[51.8, 53.199999999999996, 0],[51.099999999999994, 52.5, 0],[48.3, 52.5, 0],[47.599999999999994, 53.199999999999996, 0],[46.9, 52.5, 0],[23.099999999999998, 52.5, 0],[22.4, 53.199999999999996, 0],[21.7, 52.5, 0],[21.0, 53.199999999999996, 0],[20.299999999999997, 52.5, 0],[18.9, 52.5, 0],[17.5, 53.9, 0],[17.5, 57.4, 0],[18.2, 58.099999999999994, 0],[22.4, 58.099999999999994, 0],[21.7, 58.8, 0],[21.7, 60.199999999999996, 0],[18.2, 60.199999999999996, 0],[17.5, 60.9, 0],[17.5, 64.39999999999999, 0],[18.2, 65.1, 0],[18.9, 65.1, 0],[19.599999999999998, 65.8, 0],[20.299999999999997, 65.8, 0],[21.0, 65.1, 0],[21.7, 65.8, 0],[22.4, 65.1, 0],[23.099999999999998, 65.8, 0],[18.2, 65.8, 0],[17.5, 66.5, 0],[17.5, 70.69999999999999, 0],[18.2, 71.39999999999999, 0],[22.4, 71.39999999999999, 0],[21.7, 72.1, 0],[22.4, 72.8, 0],[21.7, 73.5, 0],[18.2, 73.5, 0],[17.5, 74.19999999999999, 0],[17.5, 77.69999999999999, 0],[18.2, 78.39999999999999, 0],[51.099999999999994, 78.39999999999999, 0],[51.099999999999994, 79.1, 0],[47.599999999999994, 79.1, 0],[46.9, 79.8, 0],[46.9, 82.6, 0],[47.599999999999994, 83.3, 0],[48.3, 82.6, 0],[49.0, 83.3, 0],[49.699999999999996, 83.3, 0],[50.4, 82.6, 0],[51.099999999999994, 83.3, 0],[51.8, 82.6, 0],[52.5, 83.3, 0],[47.599999999999994, 83.3, 0],[46.9, 84.0, 0],[46.9, 86.8, 0],[47.599999999999994, 87.5, 0],[51.099999999999994, 87.5, 0],[51.099999999999994, 89.6, 0],[47.599999999999994, 89.6, 0],[46.9, 90.3, 0],[46.9, 92.39999999999999, 0],[20.299999999999997, 92.39999999999999, 0],[18.2, 94.5, 0],[17.5, 94.5, 0],[15.399999999999999, 96.6, 0],[0.7, 96.6, 0]];
        VAR pos pos20{24} := [[81.19999999999999, 120.39999999999999, 0],[81.89999999999999, 119.69999999999999, 0],[81.89999999999999, 116.19999999999999, 0],[82.6, 115.49999999999999, 0],[82.6, 114.8, 0],[83.3, 114.1, 0],[83.3, 113.39999999999999, 0],[87.5, 109.19999999999999, 0],[88.19999999999999, 109.19999999999999, 0],[89.6, 107.8, 0],[114.1, 107.8, 0],[114.1, 130.2, 0],[88.89999999999999, 130.2, 0],[88.19999999999999, 129.5, 0],[87.5, 129.5, 0],[86.8, 128.79999999999998, 0],[86.1, 128.79999999999998, 0],[83.3, 125.99999999999999, 0],[83.3, 125.3, 0],[82.6, 124.6, 0],[82.6, 123.89999999999999, 0],[81.89999999999999, 123.19999999999999, 0],[81.89999999999999, 121.1, 0],[81.19999999999999, 120.39999999999999, 0]];
        VAR pos pos21{16} := [[58.8, 118.3, 0],[60.9, 116.19999999999999, 0],[67.19999999999999, 116.19999999999999, 0],[67.89999999999999, 116.89999999999999, 0],[71.39999999999999, 116.89999999999999, 0],[71.39999999999999, 122.49999999999999, 0],[70.0, 122.49999999999999, 0],[69.3, 123.19999999999999, 0],[68.6, 122.49999999999999, 0],[62.3, 122.49999999999999, 0],[61.599999999999994, 123.19999999999999, 0],[60.9, 123.19999999999999, 0],[60.199999999999996, 122.49999999999999, 0],[59.49999999999999, 122.49999999999999, 0],[58.8, 121.8, 0],[58.8, 118.3, 0]];
        VAR pos pos22{19} := [[58.099999999999994, 134.39999999999998, 0],[58.8, 133.7, 0],[58.8, 133.0, 0],[60.9, 130.9, 0],[67.89999999999999, 130.9, 0],[68.6, 131.6, 0],[71.39999999999999, 131.6, 0],[71.39999999999999, 137.89999999999998, 0],[70.0, 137.89999999999998, 0],[69.3, 137.2, 0],[68.6, 137.89999999999998, 0],[67.89999999999999, 137.2, 0],[62.3, 137.2, 0],[61.599999999999994, 137.89999999999998, 0],[60.9, 137.2, 0],[59.49999999999999, 137.2, 0],[58.8, 136.5, 0],[58.8, 135.1, 0],[58.099999999999994, 134.39999999999998, 0]];
        VAR pos pos23{15} := [[58.099999999999994, 105.0, 0],[58.8, 104.3, 0],[58.8, 103.6, 0],[60.199999999999996, 102.19999999999999, 0],[60.9, 102.19999999999999, 0],[61.599999999999994, 101.5, 0],[65.8, 101.5, 0],[66.5, 102.19999999999999, 0],[71.39999999999999, 102.19999999999999, 0],[71.39999999999999, 108.5, 0],[60.199999999999996, 108.5, 0],[58.8, 107.1, 0],[58.8, 106.39999999999999, 0],[58.099999999999994, 105.69999999999999, 0],[58.099999999999994, 105.0, 0]];
        VAR pos pos24{17} := [[46.9, 32.199999999999996, 0],[47.599999999999994, 31.499999999999996, 0],[47.599999999999994, 30.799999999999997, 0],[49.0, 30.799999999999997, 0],[49.699999999999996, 30.099999999999998, 0],[50.4, 30.799999999999997, 0],[53.9, 30.799999999999997, 0],[53.9, 34.3, 0],[53.199999999999996, 33.599999999999994, 0],[51.099999999999994, 33.599999999999994, 0],[50.4, 34.3, 0],[49.699999999999996, 34.3, 0],[49.0, 33.599999999999994, 0],[48.3, 34.3, 0],[47.599999999999994, 33.599999999999994, 0],[46.9, 33.599999999999994, 0],[46.9, 32.199999999999996, 0]];
        VAR pos pos25{16} := [[46.199999999999996, 207.89999999999998, 0],[47.599999999999994, 206.5, 0],[48.3, 206.5, 0],[49.0, 205.79999999999998, 0],[51.8, 205.79999999999998, 0],[52.5, 206.5, 0],[52.5, 210.0, 0],[51.8, 210.7, 0],[51.099999999999994, 210.0, 0],[50.4, 210.0, 0],[49.699999999999996, 210.7, 0],[48.3, 210.7, 0],[47.599999999999994, 210.0, 0],[46.9, 210.0, 0],[46.199999999999996, 209.29999999999998, 0],[46.199999999999996, 207.89999999999998, 0]];
        VAR pos pos26{14} := [[46.199999999999996, 174.29999999999998, 0],[47.599999999999994, 172.89999999999998, 0],[48.3, 172.89999999999998, 0],[49.0, 172.2, 0],[49.699999999999996, 172.2, 0],[50.4, 172.89999999999998, 0],[51.099999999999994, 172.89999999999998, 0],[51.8, 172.2, 0],[52.5, 172.89999999999998, 0],[52.5, 176.39999999999998, 0],[51.8, 177.1, 0],[47.599999999999994, 177.1, 0],[46.199999999999996, 175.7, 0],[46.199999999999996, 174.29999999999998, 0]];
        VAR pos pos27{16} := [[46.199999999999996, 67.89999999999999, 0],[47.599999999999994, 66.5, 0],[48.3, 66.5, 0],[49.0, 65.8, 0],[51.8, 65.8, 0],[52.5, 66.5, 0],[52.5, 70.0, 0],[51.8, 70.69999999999999, 0],[51.099999999999994, 70.0, 0],[50.4, 70.0, 0],[49.699999999999996, 70.69999999999999, 0],[48.3, 70.69999999999999, 0],[47.599999999999994, 70.0, 0],[46.9, 70.0, 0],[46.199999999999996, 69.3, 0],[46.199999999999996, 67.89999999999999, 0]];
        VAR pos pos28{15} := [[33.599999999999994, 207.2, 0],[34.3, 206.5, 0],[35.0, 206.5, 0],[35.699999999999996, 205.79999999999998, 0],[39.199999999999996, 205.79999999999998, 0],[39.199999999999996, 207.89999999999998, 0],[39.9, 208.6, 0],[39.199999999999996, 209.29999999999998, 0],[39.9, 210.0, 0],[37.8, 210.0, 0],[37.099999999999994, 210.7, 0],[35.0, 210.7, 0],[34.3, 210.0, 0],[33.599999999999994, 210.0, 0],[33.599999999999994, 207.2, 0]];
        VAR pos pos29{14} := [[33.599999999999994, 173.6, 0],[34.3, 172.89999999999998, 0],[36.4, 172.89999999999998, 0],[37.099999999999994, 172.2, 0],[37.8, 172.89999999999998, 0],[39.199999999999996, 172.89999999999998, 0],[39.199999999999996, 174.29999999999998, 0],[39.9, 175.0, 0],[39.199999999999996, 175.7, 0],[39.199999999999996, 177.1, 0],[35.0, 177.1, 0],[34.3, 176.39999999999998, 0],[33.599999999999994, 176.39999999999998, 0],[33.599999999999994, 173.6, 0]];
        VAR pos pos30{13} := [[33.599999999999994, 67.19999999999999, 0],[35.0, 65.8, 0],[35.699999999999996, 65.8, 0],[36.4, 65.1, 0],[37.099999999999994, 65.8, 0],[40.599999999999994, 65.8, 0],[41.3, 66.5, 0],[41.3, 67.89999999999999, 0],[40.599999999999994, 68.6, 0],[40.599999999999994, 69.3, 0],[39.9, 68.6, 0],[33.599999999999994, 68.6, 0],[33.599999999999994, 67.19999999999999, 0]];
        VAR pos pos31{10} := [[33.599999999999994, 32.199999999999996, 0],[35.0, 30.799999999999997, 0],[35.699999999999996, 30.799999999999997, 0],[36.4, 30.099999999999998, 0],[37.099999999999994, 30.799999999999997, 0],[40.599999999999994, 30.799999999999997, 0],[40.599999999999994, 32.9, 0],[41.3, 33.599999999999994, 0],[33.599999999999994, 33.599999999999994, 0],[33.599999999999994, 32.199999999999996, 0]];
        VAR pos pos32{23} := [[29.4, 133.0, 0],[30.799999999999997, 131.6, 0],[31.499999999999996, 131.6, 0],[32.199999999999996, 130.9, 0],[38.5, 130.9, 0],[39.199999999999996, 131.6, 0],[42.0, 131.6, 0],[42.0, 133.0, 0],[42.699999999999996, 133.7, 0],[42.0, 134.39999999999998, 0],[42.699999999999996, 135.1, 0],[42.699999999999996, 137.2, 0],[42.0, 137.2, 0],[41.3, 137.89999999999998, 0],[40.599999999999994, 137.2, 0],[34.3, 137.2, 0],[33.599999999999994, 137.89999999999998, 0],[32.9, 137.89999999999998, 0],[32.199999999999996, 137.2, 0],[30.099999999999998, 137.2, 0],[30.099999999999998, 136.5, 0],[29.4, 135.79999999999998, 0],[29.4, 133.0, 0]];
        VAR pos pos33{27} := [[29.4, 118.99999999999999, 0],[30.099999999999998, 118.3, 0],[30.099999999999998, 117.6, 0],[30.799999999999997, 116.89999999999999, 0],[31.499999999999996, 116.89999999999999, 0],[32.199999999999996, 116.19999999999999, 0],[38.5, 116.19999999999999, 0],[39.199999999999996, 116.89999999999999, 0],[42.0, 116.89999999999999, 0],[42.0, 118.99999999999999, 0],[42.699999999999996, 119.69999999999999, 0],[42.0, 120.39999999999999, 0],[42.699999999999996, 121.1, 0],[42.699999999999996, 121.8, 0],[42.0, 122.49999999999999, 0],[41.3, 122.49999999999999, 0],[40.599999999999994, 123.19999999999999, 0],[39.9, 122.49999999999999, 0],[35.0, 122.49999999999999, 0],[34.3, 123.19999999999999, 0],[33.599999999999994, 122.49999999999999, 0],[32.199999999999996, 122.49999999999999, 0],[31.499999999999996, 123.19999999999999, 0],[30.799999999999997, 122.49999999999999, 0],[30.099999999999998, 122.49999999999999, 0],[29.4, 121.8, 0],[29.4, 118.99999999999999, 0]];
        VAR pos pos34{16} := [[29.4, 104.3, 0],[30.099999999999998, 103.6, 0],[30.099999999999998, 102.89999999999999, 0],[30.799999999999997, 102.19999999999999, 0],[31.499999999999996, 102.19999999999999, 0],[32.199999999999996, 101.5, 0],[37.099999999999994, 101.5, 0],[37.8, 102.19999999999999, 0],[41.3, 102.19999999999999, 0],[42.0, 102.89999999999999, 0],[42.0, 108.5, 0],[31.499999999999996, 108.5, 0],[30.799999999999997, 107.8, 0],[30.099999999999998, 107.8, 0],[29.4, 107.1, 0],[29.4, 104.3, 0]];

        ! Define variables to be used while drawing
        VAR num font_size := 1.0;
        VAR pos position := [0,0,0];
        VAR robtarget next_target := [[0,0,0],[0,0,1,0],[0,0,0,0],[9E+09,9E+09,9E+09,9E+09,9E+09,9E+09]];

        ! Update the penup_offset based on the z_offset
        penup_offset := z_offset + penup_offset;

        ! Raise pen to avoid drawing of surface while moving to the new approach position
        position := pos0{1} * font_size;
        next_target.trans := position;
        MoveJ Offs(next_target, x_offset, y_offset, penup_offset),approach_speed,fine,Alex_Pen_ABB\WObj:=WorkSurface;

        ! Drop pen
        MoveL Offs(next_target, x_offset, y_offset, z_offset),approach_speed,fine,Alex_Pen_ABB\WObj:=WorkSurface;

        FOR index FROM 1 TO Dim(pos0, 1) DO
            position := pos0{index} * font_size;
            next_target.trans := position;

            MoveL Offs(next_target, x_offset, y_offset, z_offset),write_speed,fine,Alex_Pen_ABB\WObj:=WorkSurface;
        ENDFOR

        ! Raise pen
        MoveL Offs(next_target, x_offset, y_offset, penup_offset),approach_speed,fine,Alex_Pen_ABB\WObj:=WorkSurface;

        ! Raise pen to avoid drawing of surface while moving to the new approach position
        position := pos1{1} * font_size;
        next_target.trans := position;
        MoveJ Offs(next_target, x_offset, y_offset, penup_offset),approach_speed,fine,Alex_Pen_ABB\WObj:=WorkSurface;

        ! Drop pen
        MoveL Offs(next_target, x_offset, y_offset, z_offset),approach_speed,fine,Alex_Pen_ABB\WObj:=WorkSurface;

        FOR index FROM 1 TO Dim(pos1, 1) DO
            position := pos1{index} * font_size;
            next_target.trans := position;

            MoveL Offs(next_target, x_offset, y_offset, z_offset),write_speed,fine,Alex_Pen_ABB\WObj:=WorkSurface;
        ENDFOR

        ! Raise pen
        MoveL Offs(next_target, x_offset, y_offset, penup_offset),approach_speed,fine,Alex_Pen_ABB\WObj:=WorkSurface;

        ! Raise pen to avoid drawing of surface while moving to the new approach position
        position := pos2{1} * font_size;
        next_target.trans := position;
        MoveJ Offs(next_target, x_offset, y_offset, penup_offset),approach_speed,fine,Alex_Pen_ABB\WObj:=WorkSurface;

        ! Drop pen
        MoveL Offs(next_target, x_offset, y_offset, z_offset),approach_speed,fine,Alex_Pen_ABB\WObj:=WorkSurface;

        FOR index FROM 1 TO Dim(pos2, 1) DO
            position := pos2{index} * font_size;
            next_target.trans := position;

            MoveL Offs(next_target, x_offset, y_offset, z_offset),write_speed,fine,Alex_Pen_ABB\WObj:=WorkSurface;
        ENDFOR

        ! Raise pen
        MoveL Offs(next_target, x_offset, y_offset, penup_offset),approach_speed,fine,Alex_Pen_ABB\WObj:=WorkSurface;

        ! Raise pen to avoid drawing of surface while moving to the new approach position
        position := pos3{1} * font_size;
        next_target.trans := position;
        MoveJ Offs(next_target, x_offset, y_offset, penup_offset),approach_speed,fine,Alex_Pen_ABB\WObj:=WorkSurface;

        ! Drop pen
        MoveL Offs(next_target, x_offset, y_offset, z_offset),approach_speed,fine,Alex_Pen_ABB\WObj:=WorkSurface;

        FOR index FROM 1 TO Dim(pos3, 1) DO
            position := pos3{index} * font_size;
            next_target.trans := position;

            MoveL Offs(next_target, x_offset, y_offset, z_offset),write_speed,fine,Alex_Pen_ABB\WObj:=WorkSurface;
        ENDFOR

        ! Raise pen
        MoveL Offs(next_target, x_offset, y_offset, penup_offset),approach_speed,fine,Alex_Pen_ABB\WObj:=WorkSurface;

        ! Raise pen to avoid drawing of surface while moving to the new approach position
        position := pos4{1} * font_size;
        next_target.trans := position;
        MoveJ Offs(next_target, x_offset, y_offset, penup_offset),approach_speed,fine,Alex_Pen_ABB\WObj:=WorkSurface;

        ! Drop pen
        MoveL Offs(next_target, x_offset, y_offset, z_offset),approach_speed,fine,Alex_Pen_ABB\WObj:=WorkSurface;

        FOR index FROM 1 TO Dim(pos4, 1) DO
            position := pos4{index} * font_size;
            next_target.trans := position;

            MoveL Offs(next_target, x_offset, y_offset, z_offset),write_speed,fine,Alex_Pen_ABB\WObj:=WorkSurface;
        ENDFOR

        ! Raise pen
        MoveL Offs(next_target, x_offset, y_offset, penup_offset),approach_speed,fine,Alex_Pen_ABB\WObj:=WorkSurface;

        ! Raise pen to avoid drawing of surface while moving to the new approach position
        position := pos5{1} * font_size;
        next_target.trans := position;
        MoveJ Offs(next_target, x_offset, y_offset, penup_offset),approach_speed,fine,Alex_Pen_ABB\WObj:=WorkSurface;

        ! Drop pen
        MoveL Offs(next_target, x_offset, y_offset, z_offset),approach_speed,fine,Alex_Pen_ABB\WObj:=WorkSurface;

        FOR index FROM 1 TO Dim(pos5, 1) DO
            position := pos5{index} * font_size;
            next_target.trans := position;

            MoveL Offs(next_target, x_offset, y_offset, z_offset),write_speed,fine,Alex_Pen_ABB\WObj:=WorkSurface;
        ENDFOR

        ! Raise pen
        MoveL Offs(next_target, x_offset, y_offset, penup_offset),approach_speed,fine,Alex_Pen_ABB\WObj:=WorkSurface;

        ! Raise pen to avoid drawing of surface while moving to the new approach position
        position := pos6{1} * font_size;
        next_target.trans := position;
        MoveJ Offs(next_target, x_offset, y_offset, penup_offset),approach_speed,fine,Alex_Pen_ABB\WObj:=WorkSurface;

        ! Drop pen
        MoveL Offs(next_target, x_offset, y_offset, z_offset),approach_speed,fine,Alex_Pen_ABB\WObj:=WorkSurface;

        FOR index FROM 1 TO Dim(pos6, 1) DO
            position := pos6{index} * font_size;
            next_target.trans := position;

            MoveL Offs(next_target, x_offset, y_offset, z_offset),write_speed,fine,Alex_Pen_ABB\WObj:=WorkSurface;
        ENDFOR

        ! Raise pen
        MoveL Offs(next_target, x_offset, y_offset, penup_offset),approach_speed,fine,Alex_Pen_ABB\WObj:=WorkSurface;

        ! Raise pen to avoid drawing of surface while moving to the new approach position
        position := pos7{1} * font_size;
        next_target.trans := position;
        MoveJ Offs(next_target, x_offset, y_offset, penup_offset),approach_speed,fine,Alex_Pen_ABB\WObj:=WorkSurface;

        ! Drop pen
        MoveL Offs(next_target, x_offset, y_offset, z_offset),approach_speed,fine,Alex_Pen_ABB\WObj:=WorkSurface;

        FOR index FROM 1 TO Dim(pos7, 1) DO
            position := pos7{index} * font_size;
            next_target.trans := position;

            MoveL Offs(next_target, x_offset, y_offset, z_offset),write_speed,fine,Alex_Pen_ABB\WObj:=WorkSurface;
        ENDFOR

        ! Raise pen
        MoveL Offs(next_target, x_offset, y_offset, penup_offset),approach_speed,fine,Alex_Pen_ABB\WObj:=WorkSurface;

        ! Raise pen to avoid drawing of surface while moving to the new approach position
        position := pos8{1} * font_size;
        next_target.trans := position;
        MoveJ Offs(next_target, x_offset, y_offset, penup_offset),approach_speed,fine,Alex_Pen_ABB\WObj:=WorkSurface;

        ! Drop pen
        MoveL Offs(next_target, x_offset, y_offset, z_offset),approach_speed,fine,Alex_Pen_ABB\WObj:=WorkSurface;

        FOR index FROM 1 TO Dim(pos8, 1) DO
            position := pos8{index} * font_size;
            next_target.trans := position;

            MoveL Offs(next_target, x_offset, y_offset, z_offset),write_speed,fine,Alex_Pen_ABB\WObj:=WorkSurface;
        ENDFOR

        ! Raise pen
        MoveL Offs(next_target, x_offset, y_offset, penup_offset),approach_speed,fine,Alex_Pen_ABB\WObj:=WorkSurface;

        ! Raise pen to avoid drawing of surface while moving to the new approach position
        position := pos9{1} * font_size;
        next_target.trans := position;
        MoveJ Offs(next_target, x_offset, y_offset, penup_offset),approach_speed,fine,Alex_Pen_ABB\WObj:=WorkSurface;

        ! Drop pen
        MoveL Offs(next_target, x_offset, y_offset, z_offset),approach_speed,fine,Alex_Pen_ABB\WObj:=WorkSurface;

        FOR index FROM 1 TO Dim(pos9, 1) DO
            position := pos9{index} * font_size;
            next_target.trans := position;

            MoveL Offs(next_target, x_offset, y_offset, z_offset),write_speed,fine,Alex_Pen_ABB\WObj:=WorkSurface;
        ENDFOR

        ! Raise pen
        MoveL Offs(next_target, x_offset, y_offset, penup_offset),approach_speed,fine,Alex_Pen_ABB\WObj:=WorkSurface;

        ! Raise pen to avoid drawing of surface while moving to the new approach position
        position := pos10{1} * font_size;
        next_target.trans := position;
        MoveJ Offs(next_target, x_offset, y_offset, penup_offset),approach_speed,fine,Alex_Pen_ABB\WObj:=WorkSurface;

        ! Drop pen
        MoveL Offs(next_target, x_offset, y_offset, z_offset),approach_speed,fine,Alex_Pen_ABB\WObj:=WorkSurface;

        FOR index FROM 1 TO Dim(pos10, 1) DO
            position := pos10{index} * font_size;
            next_target.trans := position;

            MoveL Offs(next_target, x_offset, y_offset, z_offset),write_speed,fine,Alex_Pen_ABB\WObj:=WorkSurface;
        ENDFOR

        ! Raise pen
        MoveL Offs(next_target, x_offset, y_offset, penup_offset),approach_speed,fine,Alex_Pen_ABB\WObj:=WorkSurface;

        ! Raise pen to avoid drawing of surface while moving to the new approach position
        position := pos11{1} * font_size;
        next_target.trans := position;
        MoveJ Offs(next_target, x_offset, y_offset, penup_offset),approach_speed,fine,Alex_Pen_ABB\WObj:=WorkSurface;

        ! Drop pen
        MoveL Offs(next_target, x_offset, y_offset, z_offset),approach_speed,fine,Alex_Pen_ABB\WObj:=WorkSurface;

        FOR index FROM 1 TO Dim(pos11, 1) DO
            position := pos11{index} * font_size;
            next_target.trans := position;

            MoveL Offs(next_target, x_offset, y_offset, z_offset),write_speed,fine,Alex_Pen_ABB\WObj:=WorkSurface;
        ENDFOR

        ! Raise pen
        MoveL Offs(next_target, x_offset, y_offset, penup_offset),approach_speed,fine,Alex_Pen_ABB\WObj:=WorkSurface;

        ! Raise pen to avoid drawing of surface while moving to the new approach position
        position := pos12{1} * font_size;
        next_target.trans := position;
        MoveJ Offs(next_target, x_offset, y_offset, penup_offset),approach_speed,fine,Alex_Pen_ABB\WObj:=WorkSurface;

        ! Drop pen
        MoveL Offs(next_target, x_offset, y_offset, z_offset),approach_speed,fine,Alex_Pen_ABB\WObj:=WorkSurface;

        FOR index FROM 1 TO Dim(pos12, 1) DO
            position := pos12{index} * font_size;
            next_target.trans := position;

            MoveL Offs(next_target, x_offset, y_offset, z_offset),write_speed,fine,Alex_Pen_ABB\WObj:=WorkSurface;
        ENDFOR

        ! Raise pen
        MoveL Offs(next_target, x_offset, y_offset, penup_offset),approach_speed,fine,Alex_Pen_ABB\WObj:=WorkSurface;

        ! Raise pen to avoid drawing of surface while moving to the new approach position
        position := pos13{1} * font_size;
        next_target.trans := position;
        MoveJ Offs(next_target, x_offset, y_offset, penup_offset),approach_speed,fine,Alex_Pen_ABB\WObj:=WorkSurface;

        ! Drop pen
        MoveL Offs(next_target, x_offset, y_offset, z_offset),approach_speed,fine,Alex_Pen_ABB\WObj:=WorkSurface;

        FOR index FROM 1 TO Dim(pos13, 1) DO
            position := pos13{index} * font_size;
            next_target.trans := position;

            MoveL Offs(next_target, x_offset, y_offset, z_offset),write_speed,fine,Alex_Pen_ABB\WObj:=WorkSurface;
        ENDFOR

        ! Raise pen
        MoveL Offs(next_target, x_offset, y_offset, penup_offset),approach_speed,fine,Alex_Pen_ABB\WObj:=WorkSurface;

        ! Raise pen to avoid drawing of surface while moving to the new approach position
        position := pos14{1} * font_size;
        next_target.trans := position;
        MoveJ Offs(next_target, x_offset, y_offset, penup_offset),approach_speed,fine,Alex_Pen_ABB\WObj:=WorkSurface;

        ! Drop pen
        MoveL Offs(next_target, x_offset, y_offset, z_offset),approach_speed,fine,Alex_Pen_ABB\WObj:=WorkSurface;

        FOR index FROM 1 TO Dim(pos14, 1) DO
            position := pos14{index} * font_size;
            next_target.trans := position;

            MoveL Offs(next_target, x_offset, y_offset, z_offset),write_speed,fine,Alex_Pen_ABB\WObj:=WorkSurface;
        ENDFOR

        ! Raise pen
        MoveL Offs(next_target, x_offset, y_offset, penup_offset),approach_speed,fine,Alex_Pen_ABB\WObj:=WorkSurface;

        ! Raise pen to avoid drawing of surface while moving to the new approach position
        position := pos15{1} * font_size;
        next_target.trans := position;
        MoveJ Offs(next_target, x_offset, y_offset, penup_offset),approach_speed,fine,Alex_Pen_ABB\WObj:=WorkSurface;

        ! Drop pen
        MoveL Offs(next_target, x_offset, y_offset, z_offset),approach_speed,fine,Alex_Pen_ABB\WObj:=WorkSurface;

        FOR index FROM 1 TO Dim(pos15, 1) DO
            position := pos15{index} * font_size;
            next_target.trans := position;

            MoveL Offs(next_target, x_offset, y_offset, z_offset),write_speed,fine,Alex_Pen_ABB\WObj:=WorkSurface;
        ENDFOR

        ! Raise pen
        MoveL Offs(next_target, x_offset, y_offset, penup_offset),approach_speed,fine,Alex_Pen_ABB\WObj:=WorkSurface;

        ! Raise pen to avoid drawing of surface while moving to the new approach position
        position := pos16{1} * font_size;
        next_target.trans := position;
        MoveJ Offs(next_target, x_offset, y_offset, penup_offset),approach_speed,fine,Alex_Pen_ABB\WObj:=WorkSurface;

        ! Drop pen
        MoveL Offs(next_target, x_offset, y_offset, z_offset),approach_speed,fine,Alex_Pen_ABB\WObj:=WorkSurface;

        FOR index FROM 1 TO Dim(pos16, 1) DO
            position := pos16{index} * font_size;
            next_target.trans := position;

            MoveL Offs(next_target, x_offset, y_offset, z_offset),write_speed,fine,Alex_Pen_ABB\WObj:=WorkSurface;
        ENDFOR

        ! Raise pen
        MoveL Offs(next_target, x_offset, y_offset, penup_offset),approach_speed,fine,Alex_Pen_ABB\WObj:=WorkSurface;

        ! Raise pen to avoid drawing of surface while moving to the new approach position
        position := pos17{1} * font_size;
        next_target.trans := position;
        MoveJ Offs(next_target, x_offset, y_offset, penup_offset),approach_speed,fine,Alex_Pen_ABB\WObj:=WorkSurface;

        ! Drop pen
        MoveL Offs(next_target, x_offset, y_offset, z_offset),approach_speed,fine,Alex_Pen_ABB\WObj:=WorkSurface;

        FOR index FROM 1 TO Dim(pos17, 1) DO
            position := pos17{index} * font_size;
            next_target.trans := position;

            MoveL Offs(next_target, x_offset, y_offset, z_offset),write_speed,fine,Alex_Pen_ABB\WObj:=WorkSurface;
        ENDFOR

        ! Raise pen
        MoveL Offs(next_target, x_offset, y_offset, penup_offset),approach_speed,fine,Alex_Pen_ABB\WObj:=WorkSurface;

        ! Raise pen to avoid drawing of surface while moving to the new approach position
        position := pos18{1} * font_size;
        next_target.trans := position;
        MoveJ Offs(next_target, x_offset, y_offset, penup_offset),approach_speed,fine,Alex_Pen_ABB\WObj:=WorkSurface;

        ! Drop pen
        MoveL Offs(next_target, x_offset, y_offset, z_offset),approach_speed,fine,Alex_Pen_ABB\WObj:=WorkSurface;

        FOR index FROM 1 TO Dim(pos18, 1) DO
            position := pos18{index} * font_size;
            next_target.trans := position;

            MoveL Offs(next_target, x_offset, y_offset, z_offset),write_speed,fine,Alex_Pen_ABB\WObj:=WorkSurface;
        ENDFOR

        ! Raise pen
        MoveL Offs(next_target, x_offset, y_offset, penup_offset),approach_speed,fine,Alex_Pen_ABB\WObj:=WorkSurface;

        ! Raise pen to avoid drawing of surface while moving to the new approach position
        position := pos19{1} * font_size;
        next_target.trans := position;
        MoveJ Offs(next_target, x_offset, y_offset, penup_offset),approach_speed,fine,Alex_Pen_ABB\WObj:=WorkSurface;

        ! Drop pen
        MoveL Offs(next_target, x_offset, y_offset, z_offset),approach_speed,fine,Alex_Pen_ABB\WObj:=WorkSurface;

        FOR index FROM 1 TO Dim(pos19, 1) DO
            position := pos19{index} * font_size;
            next_target.trans := position;

            MoveL Offs(next_target, x_offset, y_offset, z_offset),write_speed,fine,Alex_Pen_ABB\WObj:=WorkSurface;
        ENDFOR

        ! Raise pen
        MoveL Offs(next_target, x_offset, y_offset, penup_offset),approach_speed,fine,Alex_Pen_ABB\WObj:=WorkSurface;

        ! Raise pen to avoid drawing of surface while moving to the new approach position
        position := pos20{1} * font_size;
        next_target.trans := position;
        MoveJ Offs(next_target, x_offset, y_offset, penup_offset),approach_speed,fine,Alex_Pen_ABB\WObj:=WorkSurface;

        ! Drop pen
        MoveL Offs(next_target, x_offset, y_offset, z_offset),approach_speed,fine,Alex_Pen_ABB\WObj:=WorkSurface;

        FOR index FROM 1 TO Dim(pos20, 1) DO
            position := pos20{index} * font_size;
            next_target.trans := position;

            MoveL Offs(next_target, x_offset, y_offset, z_offset),write_speed,fine,Alex_Pen_ABB\WObj:=WorkSurface;
        ENDFOR

        ! Raise pen
        MoveL Offs(next_target, x_offset, y_offset, penup_offset),approach_speed,fine,Alex_Pen_ABB\WObj:=WorkSurface;

        ! Raise pen to avoid drawing of surface while moving to the new approach position
        position := pos21{1} * font_size;
        next_target.trans := position;
        MoveJ Offs(next_target, x_offset, y_offset, penup_offset),approach_speed,fine,Alex_Pen_ABB\WObj:=WorkSurface;

        ! Drop pen
        MoveL Offs(next_target, x_offset, y_offset, z_offset),approach_speed,fine,Alex_Pen_ABB\WObj:=WorkSurface;

        FOR index FROM 1 TO Dim(pos21, 1) DO
            position := pos21{index} * font_size;
            next_target.trans := position;

            MoveL Offs(next_target, x_offset, y_offset, z_offset),write_speed,fine,Alex_Pen_ABB\WObj:=WorkSurface;
        ENDFOR

        ! Raise pen
        MoveL Offs(next_target, x_offset, y_offset, penup_offset),approach_speed,fine,Alex_Pen_ABB\WObj:=WorkSurface;

        ! Raise pen to avoid drawing of surface while moving to the new approach position
        position := pos22{1} * font_size;
        next_target.trans := position;
        MoveJ Offs(next_target, x_offset, y_offset, penup_offset),approach_speed,fine,Alex_Pen_ABB\WObj:=WorkSurface;

        ! Drop pen
        MoveL Offs(next_target, x_offset, y_offset, z_offset),approach_speed,fine,Alex_Pen_ABB\WObj:=WorkSurface;

        FOR index FROM 1 TO Dim(pos22, 1) DO
            position := pos22{index} * font_size;
            next_target.trans := position;

            MoveL Offs(next_target, x_offset, y_offset, z_offset),write_speed,fine,Alex_Pen_ABB\WObj:=WorkSurface;
        ENDFOR

        ! Raise pen
        MoveL Offs(next_target, x_offset, y_offset, penup_offset),approach_speed,fine,Alex_Pen_ABB\WObj:=WorkSurface;

        ! Raise pen to avoid drawing of surface while moving to the new approach position
        position := pos23{1} * font_size;
        next_target.trans := position;
        MoveJ Offs(next_target, x_offset, y_offset, penup_offset),approach_speed,fine,Alex_Pen_ABB\WObj:=WorkSurface;

        ! Drop pen
        MoveL Offs(next_target, x_offset, y_offset, z_offset),approach_speed,fine,Alex_Pen_ABB\WObj:=WorkSurface;

        FOR index FROM 1 TO Dim(pos23, 1) DO
            position := pos23{index} * font_size;
            next_target.trans := position;

            MoveL Offs(next_target, x_offset, y_offset, z_offset),write_speed,fine,Alex_Pen_ABB\WObj:=WorkSurface;
        ENDFOR

        ! Raise pen
        MoveL Offs(next_target, x_offset, y_offset, penup_offset),approach_speed,fine,Alex_Pen_ABB\WObj:=WorkSurface;

        ! Raise pen to avoid drawing of surface while moving to the new approach position
        position := pos24{1} * font_size;
        next_target.trans := position;
        MoveJ Offs(next_target, x_offset, y_offset, penup_offset),approach_speed,fine,Alex_Pen_ABB\WObj:=WorkSurface;

        ! Drop pen
        MoveL Offs(next_target, x_offset, y_offset, z_offset),approach_speed,fine,Alex_Pen_ABB\WObj:=WorkSurface;

        FOR index FROM 1 TO Dim(pos24, 1) DO
            position := pos24{index} * font_size;
            next_target.trans := position;

            MoveL Offs(next_target, x_offset, y_offset, z_offset),write_speed,fine,Alex_Pen_ABB\WObj:=WorkSurface;
        ENDFOR

        ! Raise pen
        MoveL Offs(next_target, x_offset, y_offset, penup_offset),approach_speed,fine,Alex_Pen_ABB\WObj:=WorkSurface;

        ! Raise pen to avoid drawing of surface while moving to the new approach position
        position := pos25{1} * font_size;
        next_target.trans := position;
        MoveJ Offs(next_target, x_offset, y_offset, penup_offset),approach_speed,fine,Alex_Pen_ABB\WObj:=WorkSurface;

        ! Drop pen
        MoveL Offs(next_target, x_offset, y_offset, z_offset),approach_speed,fine,Alex_Pen_ABB\WObj:=WorkSurface;

        FOR index FROM 1 TO Dim(pos25, 1) DO
            position := pos25{index} * font_size;
            next_target.trans := position;

            MoveL Offs(next_target, x_offset, y_offset, z_offset),write_speed,fine,Alex_Pen_ABB\WObj:=WorkSurface;
        ENDFOR

        ! Raise pen
        MoveL Offs(next_target, x_offset, y_offset, penup_offset),approach_speed,fine,Alex_Pen_ABB\WObj:=WorkSurface;

        ! Raise pen to avoid drawing of surface while moving to the new approach position
        position := pos26{1} * font_size;
        next_target.trans := position;
        MoveJ Offs(next_target, x_offset, y_offset, penup_offset),approach_speed,fine,Alex_Pen_ABB\WObj:=WorkSurface;

        ! Drop pen
        MoveL Offs(next_target, x_offset, y_offset, z_offset),approach_speed,fine,Alex_Pen_ABB\WObj:=WorkSurface;

        FOR index FROM 1 TO Dim(pos26, 1) DO
            position := pos26{index} * font_size;
            next_target.trans := position;

            MoveL Offs(next_target, x_offset, y_offset, z_offset),write_speed,fine,Alex_Pen_ABB\WObj:=WorkSurface;
        ENDFOR

        ! Raise pen
        MoveL Offs(next_target, x_offset, y_offset, penup_offset),approach_speed,fine,Alex_Pen_ABB\WObj:=WorkSurface;

        ! Raise pen to avoid drawing of surface while moving to the new approach position
        position := pos27{1} * font_size;
        next_target.trans := position;
        MoveJ Offs(next_target, x_offset, y_offset, penup_offset),approach_speed,fine,Alex_Pen_ABB\WObj:=WorkSurface;

        ! Drop pen
        MoveL Offs(next_target, x_offset, y_offset, z_offset),approach_speed,fine,Alex_Pen_ABB\WObj:=WorkSurface;

        FOR index FROM 1 TO Dim(pos27, 1) DO
            position := pos27{index} * font_size;
            next_target.trans := position;

            MoveL Offs(next_target, x_offset, y_offset, z_offset),write_speed,fine,Alex_Pen_ABB\WObj:=WorkSurface;
        ENDFOR

        ! Raise pen
        MoveL Offs(next_target, x_offset, y_offset, penup_offset),approach_speed,fine,Alex_Pen_ABB\WObj:=WorkSurface;

        ! Raise pen to avoid drawing of surface while moving to the new approach position
        position := pos28{1} * font_size;
        next_target.trans := position;
        MoveJ Offs(next_target, x_offset, y_offset, penup_offset),approach_speed,fine,Alex_Pen_ABB\WObj:=WorkSurface;

        ! Drop pen
        MoveL Offs(next_target, x_offset, y_offset, z_offset),approach_speed,fine,Alex_Pen_ABB\WObj:=WorkSurface;

        FOR index FROM 1 TO Dim(pos28, 1) DO
            position := pos28{index} * font_size;
            next_target.trans := position;

            MoveL Offs(next_target, x_offset, y_offset, z_offset),write_speed,fine,Alex_Pen_ABB\WObj:=WorkSurface;
        ENDFOR

        ! Raise pen
        MoveL Offs(next_target, x_offset, y_offset, penup_offset),approach_speed,fine,Alex_Pen_ABB\WObj:=WorkSurface;

        ! Raise pen to avoid drawing of surface while moving to the new approach position
        position := pos29{1} * font_size;
        next_target.trans := position;
        MoveJ Offs(next_target, x_offset, y_offset, penup_offset),approach_speed,fine,Alex_Pen_ABB\WObj:=WorkSurface;

        ! Drop pen
        MoveL Offs(next_target, x_offset, y_offset, z_offset),approach_speed,fine,Alex_Pen_ABB\WObj:=WorkSurface;

        FOR index FROM 1 TO Dim(pos29, 1) DO
            position := pos29{index} * font_size;
            next_target.trans := position;

            MoveL Offs(next_target, x_offset, y_offset, z_offset),write_speed,fine,Alex_Pen_ABB\WObj:=WorkSurface;
        ENDFOR

        ! Raise pen
        MoveL Offs(next_target, x_offset, y_offset, penup_offset),approach_speed,fine,Alex_Pen_ABB\WObj:=WorkSurface;

        ! Raise pen to avoid drawing of surface while moving to the new approach position
        position := pos30{1} * font_size;
        next_target.trans := position;
        MoveJ Offs(next_target, x_offset, y_offset, penup_offset),approach_speed,fine,Alex_Pen_ABB\WObj:=WorkSurface;

        ! Drop pen
        MoveL Offs(next_target, x_offset, y_offset, z_offset),approach_speed,fine,Alex_Pen_ABB\WObj:=WorkSurface;

        FOR index FROM 1 TO Dim(pos30, 1) DO
            position := pos30{index} * font_size;
            next_target.trans := position;

            MoveL Offs(next_target, x_offset, y_offset, z_offset),write_speed,fine,Alex_Pen_ABB\WObj:=WorkSurface;
        ENDFOR

        ! Raise pen
        MoveL Offs(next_target, x_offset, y_offset, penup_offset),approach_speed,fine,Alex_Pen_ABB\WObj:=WorkSurface;

        ! Raise pen to avoid drawing of surface while moving to the new approach position
        position := pos31{1} * font_size;
        next_target.trans := position;
        MoveJ Offs(next_target, x_offset, y_offset, penup_offset),approach_speed,fine,Alex_Pen_ABB\WObj:=WorkSurface;

        ! Drop pen
        MoveL Offs(next_target, x_offset, y_offset, z_offset),approach_speed,fine,Alex_Pen_ABB\WObj:=WorkSurface;

        FOR index FROM 1 TO Dim(pos31, 1) DO
            position := pos31{index} * font_size;
            next_target.trans := position;

            MoveL Offs(next_target, x_offset, y_offset, z_offset),write_speed,fine,Alex_Pen_ABB\WObj:=WorkSurface;
        ENDFOR

        ! Raise pen
        MoveL Offs(next_target, x_offset, y_offset, penup_offset),approach_speed,fine,Alex_Pen_ABB\WObj:=WorkSurface;

        ! Raise pen to avoid drawing of surface while moving to the new approach position
        position := pos32{1} * font_size;
        next_target.trans := position;
        MoveJ Offs(next_target, x_offset, y_offset, penup_offset),approach_speed,fine,Alex_Pen_ABB\WObj:=WorkSurface;

        ! Drop pen
        MoveL Offs(next_target, x_offset, y_offset, z_offset),approach_speed,fine,Alex_Pen_ABB\WObj:=WorkSurface;

        FOR index FROM 1 TO Dim(pos32, 1) DO
            position := pos32{index} * font_size;
            next_target.trans := position;

            MoveL Offs(next_target, x_offset, y_offset, z_offset),write_speed,fine,Alex_Pen_ABB\WObj:=WorkSurface;
        ENDFOR

        ! Raise pen
        MoveL Offs(next_target, x_offset, y_offset, penup_offset),approach_speed,fine,Alex_Pen_ABB\WObj:=WorkSurface;

        ! Raise pen to avoid drawing of surface while moving to the new approach position
        position := pos33{1} * font_size;
        next_target.trans := position;
        MoveJ Offs(next_target, x_offset, y_offset, penup_offset),approach_speed,fine,Alex_Pen_ABB\WObj:=WorkSurface;

        ! Drop pen
        MoveL Offs(next_target, x_offset, y_offset, z_offset),approach_speed,fine,Alex_Pen_ABB\WObj:=WorkSurface;

        FOR index FROM 1 TO Dim(pos33, 1) DO
            position := pos33{index} * font_size;
            next_target.trans := position;

            MoveL Offs(next_target, x_offset, y_offset, z_offset),write_speed,fine,Alex_Pen_ABB\WObj:=WorkSurface;
        ENDFOR

        ! Raise pen
        MoveL Offs(next_target, x_offset, y_offset, penup_offset),approach_speed,fine,Alex_Pen_ABB\WObj:=WorkSurface;

        ! Raise pen to avoid drawing of surface while moving to the new approach position
        position := pos34{1} * font_size;
        next_target.trans := position;
        MoveJ Offs(next_target, x_offset, y_offset, penup_offset),approach_speed,fine,Alex_Pen_ABB\WObj:=WorkSurface;

        ! Drop pen
        MoveL Offs(next_target, x_offset, y_offset, z_offset),approach_speed,fine,Alex_Pen_ABB\WObj:=WorkSurface;

        FOR index FROM 1 TO Dim(pos34, 1) DO
            position := pos34{index} * font_size;
            next_target.trans := position;

            MoveL Offs(next_target, x_offset, y_offset, z_offset),write_speed,fine,Alex_Pen_ABB\WObj:=WorkSurface;
        ENDFOR

        ! Raise pen
        MoveL Offs(next_target, x_offset, y_offset, penup_offset),approach_speed,fine,Alex_Pen_ABB\WObj:=WorkSurface;

    ENDPROC

    !***********************************************************
    !
    ! Procedure DrawMyTextArt
    !   This procedure draws Middlezex University's LOGO on the work surface
    !
    ! Example
    !   DrawMyTextArt;
    !
    ! Warning
    !   Takes a long time to complete
    !
    !***********************************************************
    PROC DrawMyTextArt()
        VAR num font_size := 0.06;
        VAR num x_offset := 5;
        VAR num y_offset := 5;
        VAR num line_height := 50;

        line_height := line_height * font_size;

        DrawString "@@@'#@'@@@@@@@++@'@@@@@@'@;@@@@@@@@;#;@@@@@;@@@@@@@@@'@'@@@@@@@@@@'", font_size, v500, v800, x_offset, y_offset, 0, 30;
        y_offset := y_offset + line_height;
        DrawString "@@@@'';@@@@@@@@+';@@@@@@#++;@@@@@@@@@@@@@@#'@##@@@@@#@#'@@@@@@@@+@'", font_size, v500, v800, x_offset, y_offset, 0, 30;
        y_offset := y_offset + line_height;
        DrawString "@@@@@@@@@@@@@@@@@@@@@@@@#;#+#@@@@@@@@@@@@@@'++@@@@@@'@''@@@@@@@@@@@", font_size, v500, v800, x_offset, y_offset, 0, 30;
        y_offset := y_offset + line_height;
        DrawString "@@@@@@@@@@@@@@@@@@@@@@@@@+;;@@@@@@@@@@@@@@@@@@@@@@@@@'@+@@@@@@@@@@@", font_size, v500, v800, x_offset, y_offset, 0, 30;
        y_offset := y_offset + line_height;
        DrawString "@@@@@@@@@@@@@@@@@@@@@@@@@@@@@@@@@@@@@@@@@@@@@@@@@@@@@@@@@@@@@@@@@@@", font_size, v500, v800, x_offset, y_offset, 0, 30;
        y_offset := y_offset + line_height;
        DrawString "@@@@@@@@@@@@@@@@@@@@@@#++'';;;;''''';;;;''++#@@@@@@@@@@@@@@@@@@@@@@", font_size, v500, v800, x_offset, y_offset, 0, 30;
        y_offset := y_offset + line_height;
        DrawString "@@@@@@@@@@@@@@@@@@;'''''''''''''''''''''''''''''''@@@@@@@@@@#@@@@@@", font_size, v500, v800, x_offset, y_offset, 0, 30;
        y_offset := y_offset + line_height;
        DrawString "@@@@@@@@@@@#@@@@@@;'''''''''''''''''''''''''''''''@@@@@@@@@@';+@@@@", font_size, v500, v800, x_offset, y_offset, 0, 30;
        y_offset := y_offset + line_height;
        DrawString "@@@@@@@@@'#'@@@@@@''''''''''';'''@+''';'''''''''''@@@@@@@@@@'#+'@@@", font_size, v500, v800, x_offset, y_offset, 0, 30;
        y_offset := y_offset + line_height;
        DrawString "@@@@@@@@#'@'@@@@@@'''''''''''@'''@;''+@'''''''''''@@@@@@@@@@+@@'@@@", font_size, v500, v800, x_offset, y_offset, 0, 30;
        y_offset := y_offset + line_height;
        DrawString "@@@@@@@@'@@+@@@@@@'''''''''';@;''@'''##'''''''''';@@@@@@@@@@@@;:@@@", font_size, v500, v800, x_offset, y_offset, 0, 30;
        y_offset := y_offset + line_height;
        DrawString "@@@@@@@@#'+#@@@@@@''''''''''''@'#@@#'@''''''''''';@@@@@@@@@@@@@@@@@", font_size, v500, v800, x_offset, y_offset, 0, 30;
        y_offset := y_offset + line_height;
        DrawString "@@@@@@@@@;@;@@@@@@''''''''''';@@@@@@@@''''''''''';@@@@@@@@@@@@@@@@@", font_size, v500, v800, x_offset, y_offset, 0, 30;
        y_offset := y_offset + line_height;
        DrawString "@@@@@@@@@@@@@@@@@@''''''''''''@+';;'##''''''''''';@@@@@@@@@@@@@@@@@", font_size, v500, v800, x_offset, y_offset, 0, 30;
        y_offset := y_offset + line_height;
        DrawString "@@@@@@@@@@@@@@@@@@''''''''''''+#'''+@;''''''''''';@@@@@@@@@@@@@@@@@", font_size, v500, v800, x_offset, y_offset, 0, 30;
        y_offset := y_offset + line_height;
        DrawString "@@@@@@@@@@@@@@@@@@'''''''''''''';;;;''''''''''''';@@@@@@@@@@@@@@@@@", font_size, v500, v800, x_offset, y_offset, 0, 30;
        y_offset := y_offset + line_height;
        DrawString "@@@@@@@'@@@@@@@@@@;'''''''''''''''''''''''''''''''@@@;#+@@@@@@@@@@@", font_size, v500, v800, x_offset, y_offset, 0, 30;
        y_offset := y_offset + line_height;
        DrawString "@@@@@@'+;@@@@@@@@@;'''''''''''''''''''''''''''''''@@@;@'@@@@@@@@@@@", font_size, v500, v800, x_offset, y_offset, 0, 30;
        y_offset := y_offset + line_height;
        DrawString "@@@@@@'++;@@@@@@@@;''''''';+'''';;;;;''''''''''''+@@@#@;@@@@@@@@@@@", font_size, v500, v800, x_offset, y_offset, 0, 30;
        y_offset := y_offset + line_height;
        DrawString "@@@@@@+'@#;@@@@@@@''''''''#';+@@@@@@@@@+;''''''''#@@@'#+;@@@@@@@@@@", font_size, v500, v800, x_offset, y_offset, 0, 30;
        y_offset := y_offset + line_height;
        DrawString "@@@@@@@#:'@@@@@@@@+'''''';#@@@@@@@@@@@@@@@;''''''@@@@#+'@@@#'#+@@@@", font_size, v500, v800, x_offset, y_offset, 0, 30;
        y_offset := y_offset + line_height;
        DrawString "@@@@@@@@@@@@@@@@@@#'''';+@@@@+';;;'#@';@@@@''''';@@@@@@@@@@'#+;#@@@", font_size, v500, v800, x_offset, y_offset, 0, 30;
        y_offset := y_offset + line_height;
        DrawString "@@@@@@@@@@@@@@@@@@@''''@@@+#;''''''''''@@@@@'''';@@@@@@@@@@@'#@;@@@", font_size, v500, v800, x_offset, y_offset, 0, 30;
        y_offset := y_offset + line_height;
        DrawString "@@@@@@@@@@@@@@@@@@@;'';@'';@'''''''''''@@@@@@''''@@@@@@@@@@@@'#;@@@", font_size, v500, v800, x_offset, y_offset, 0, 30;
        y_offset := y_offset + line_height;
        DrawString "@@@@@@@@@@@@@@@@@@@+''''''';'''''''''''';;;;;'''@@@@@@@@@@@@@@#@@@@", font_size, v500, v800, x_offset, y_offset, 0, 30;
        y_offset := y_offset + line_height;
        DrawString "@@@@@@@@@@@@@@@@@@@@''''''''+''''';;''''''''''';@@@@@@@@@@@@@@@@@@@", font_size, v500, v800, x_offset, y_offset, 0, 30;
        y_offset := y_offset + line_height;
        DrawString "@@@@@@@@@@@@@@@@@@@@;'''''';+;+@@@@@@@+;''''''''@@@@@@@@@@@@@@@@@@@", font_size, v500, v800, x_offset, y_offset, 0, 30;
        y_offset := y_offset + line_height;
        DrawString "@@@@@@@@@@@@@@@@@@@@+''''';+@@@@@@@@@#@@#;'''''@@@@@@+#@@@@@@@@@@@@", font_size, v500, v800, x_offset, y_offset, 0, 30;
        y_offset := y_offset + line_height;
        DrawString "@@@@@@@@@@@@@@@@@@@@@''''#@@@';;';;'''@@@@;''';@@@@@'#'@@@@@@@@@@@@", font_size, v500, v800, x_offset, y_offset, 0, 30;
        y_offset := y_offset + line_height;
        DrawString "@@@@@@@@@@@@@@@@@@@@@+'''@+;@;''''''';@@@@@'''@@@@@;@#'@@@@@@@@@@@@", font_size, v500, v800, x_offset, y_offset, 0, 30;
        y_offset := y_offset + line_height;
        DrawString "@@@@''+#;@@@@@@@@@@@@@'''''';'''''''''';;;;'';@@@@#@'@;@@@@@@@@@@@@", font_size, v500, v800, x_offset, y_offset, 0, 30;
        y_offset := y_offset + line_height;
        DrawString "@@@@''@@;@@@@@@@@@@@@@#''''''''''''''''''''''@@@@@@@+##@@@@@@@@@@@@", font_size, v500, v800, x_offset, y_offset, 0, 30;
        y_offset := y_offset + line_height;
        DrawString "@@@@+++#@@@@@@@@@@@@@@@;'''''@;#@@@@#';'''''+@@@@@@@+@@@@@@@@#@@@@@", font_size, v500, v800, x_offset, y_offset, 0, 30;
        y_offset := y_offset + line_height;
        DrawString "@@@@@'#@@@@@@@@@@@@@@@@@''';+@@@@#@#'@@'''';@@@@@@@@@@@@@@@#;+@+@@@", font_size, v500, v800, x_offset, y_offset, 0, 30;
        y_offset := y_offset + line_height;
        DrawString "@@@@@@@@@@@@@@@@@@@@@@@@@''@@'+''''';@@@;';@@@@@@@@@@@@@@@@;'@#'@@@", font_size, v500, v800, x_offset, y_offset, 0, 30;
        y_offset := y_offset + line_height;
        DrawString "@@@@@@@@@@@@@';@@@@@@@@@@#';'+;'''''''''';@@@@@@@@@@@@@@@@@'##'@@@@", font_size, v500, v800, x_offset, y_offset, 0, 30;
        y_offset := y_offset + line_height;
        DrawString "@@@@@@@@@@@@++#+@@@@@@@@@@#''''''''''''';@@@@@@@@@@@@@@@@@@##+@@@@@", font_size, v500, v800, x_offset, y_offset, 0, 30;
        y_offset := y_offset + line_height;
        DrawString "@@@@@@@@@@@@;'+@@@@@@@@@@@@#''''''''''';@@@@@@@@@@@@@@@@@@@@@@@@@@@", font_size, v500, v800, x_offset, y_offset, 0, 30;
        y_offset := y_offset + line_height;
        DrawString "@@@@@@@@@@@@'+##@@@@@@@@@@@@@;'''''''''@@@@@@@@@@'@#@@@@@@@@@@@@@@@", font_size, v500, v800, x_offset, y_offset, 0, 30;
        y_offset := y_offset + line_height;
        DrawString "@@@@@@@@@@@@#'+:@@@+#@@@@@@@@@'''''';#@@@@@@@@@@#@#''@@@@@@@@@@@@@@", font_size, v500, v800, x_offset, y_offset, 0, 30;
        y_offset := y_offset + line_height;
        DrawString "@@@@@@@'@@@@@+@@@@@+@;@@@@@@@@@@;'''@@@@@@@@@@@@+'@@+@@@@@@@@@@@@@@", font_size, v500, v800, x_offset, y_offset, 0, 30;
        y_offset := y_offset + line_height;
        DrawString "@@@@@@'+;@@@@@@@@@@'@@'@@@@@@@@@@@@@@@@@@@@@@@@@@#:+;@@@@@@@@@@@@@@", font_size, v500, v800, x_offset, y_offset, 0, 30;
        y_offset := y_offset + line_height;
        DrawString "@@@@@@'++;@@@@@@@@@'@+'@@@@@@@@@@@@@@@@@@@@@@@@@@@@#@@@@@@@@@@@@@@@", font_size, v500, v800, x_offset, y_offset, 0, 30;
        y_offset := y_offset + line_height;
        DrawString "@@@@@@+'@#;@@@@@@@@'#;@@@@@@@@@@@@@@@@@@@@@@@@@@@@@@@@@@@@@@@@@@@@@", font_size, v500, v800, x_offset, y_offset, 0, 30;
        y_offset := y_offset + line_height;
        DrawString "@@@@@@@#:+@@@@@@@@@@@'@@@@@@@@@@@@@@@@@@;'@@@@@@@@@@@@@@@@@@@@@@@@@", font_size, v500, v800, x_offset, y_offset, 0, 30;
        y_offset := y_offset + line_height;
        DrawString "@@@@@@@@@@@@@@@@@@@@@@@@@@@@+@@@@@@@@@@'@#@@@@@@@@@@@@@@@@@@@@@@@@@", font_size, v500, v800, x_offset, y_offset, 0, 30;
        y_offset := y_offset + line_height;
        DrawString "@@@@@@@@@@@@@@@@@@@@@@@@@@@'+:@@@@@@@@#@''@@@@@@@@@@@@@@@@@@@@@@@@@", font_size, v500, v800, x_offset, y_offset, 0, 30;
        y_offset := y_offset + line_height;
        DrawString "@@@@@@@@@@@@@@@@@@@@@@@@@@@;@';@@@@@@@'#@;@@@@@@@@@@@@@@@@@@@@@@@@@", font_size, v500, v800, x_offset, y_offset, 0, 30;
        y_offset := y_offset + line_height;
    ENDPROC

    !***********************************************************
    !
    ! Function get_character_width
    !   This function returns the width of a given character
    !
    ! Example
    !   VAR string character_a := "a";
    !   a_width := get_character_width(character_a);
    !
    !***********************************************************
    FUNC num get_character_width(string character)
        VAR num char_width := 20;

        ! Determine the width of the character
        IF character = " " THEN
            char_width := 20;
        ELSEIF character = "!" THEN
            char_width := 10;
        ELSEIF character = """" THEN
            char_width := 22;
        ELSEIF character = "'" THEN
            char_width := 6;
        ELSEIF character = "#" THEN
            char_width := 38;
        ELSEIF character = "$" THEN
            char_width := 34;
        ELSEIF character = "%" THEN
            char_width := 42;
        ELSEIF character = "&" THEN
            char_width := 46;
        ELSEIF character = "(" THEN
            char_width := 20;
        ELSEIF character = ")" THEN
            char_width := 20;
        ELSEIF character = "*" THEN
            char_width := 26;
        ELSEIF character = "+" THEN
            char_width := 42;
        ELSEIF character = "," THEN
            char_width := 10;
        ELSEIF character = "-" THEN
            char_width := 42;
        ELSEIF character = "." THEN
            char_width := 10;
        ELSEIF character = "/" THEN
            char_width := 42;
        ELSEIF character = "0" THEN
            char_width := 34;
        ELSEIF character = "1" THEN
            char_width := 16;
        ELSEIF character = "2" THEN
            char_width := 34;
        ELSEIF character = "3" THEN
            char_width := 34;
        ELSEIF character = "4" THEN
            char_width := 36;
        ELSEIF character = "5" THEN
            char_width := 34;
        ELSEIF character = "6" THEN
            char_width := 32;
        ELSEIF character = "7" THEN
            char_width := 34;
        ELSEIF character = "8" THEN
            char_width := 34;
        ELSEIF character = "9" THEN
            char_width := 32;
        ELSEIF character = ":" THEN
            char_width := 10;
        ELSEIF character = ";" THEN
            char_width := 10;
        ELSEIF character = "<" THEN
            char_width := 38;
        ELSEIF character = ">" THEN
            char_width := 38;
        ELSEIF character = "=" THEN
            char_width := 42;
        ELSEIF character = "?" THEN
            char_width := 30;
        ELSEIF character = "@" THEN
            char_width := 48;
        ELSEIF character = "A" THEN
            char_width := 38;
        ELSEIF character = "B" THEN
            char_width := 34;
        ELSEIF character = "C" THEN
            char_width := 36;
        ELSEIF character = "D" THEN
            char_width := 34;
        ELSEIF character = "E" THEN
            char_width := 32;
        ELSEIF character = "F" THEN
            char_width := 32;
        ELSEIF character = "G" THEN
            char_width := 36;
        ELSEIF character = "H" THEN
            char_width := 34;
        ELSEIF character = "I" THEN
            char_width := 6;
        ELSEIF character = "J" THEN
            char_width := 26;
        ELSEIF character = "K" THEN
            char_width := 34;
        ELSEIF character = "L" THEN
            char_width := 30;
        ELSEIF character = "M" THEN
            char_width := 38;
        ELSEIF character = "N" THEN
            char_width := 34;
        ELSEIF character = "O" THEN
            char_width := 38;
        ELSEIF character = "P" THEN
            char_width := 34;
        ELSEIF character = "Q" THEN
            char_width := 38;
        ELSEIF character = "R" THEN
            char_width := 34;
        ELSEIF character = "S" THEN
            char_width := 34;
        ELSEIF character = "T" THEN
            char_width := 34;
        ELSEIF character = "U" THEN
            char_width := 34;
        ELSEIF character = "V" THEN
            char_width := 38;
        ELSEIF character = "W" THEN
            char_width := 46;
        ELSEIF character = "X" THEN
            char_width := 34;
        ELSEIF character = "Y" THEN
            char_width := 38;
        ELSEIF character = "Z" THEN
            char_width := 34;
        ELSEIF character = "[" THEN
            char_width := 20;
        ELSEIF character = "]" THEN
            char_width := 20;
        ELSEIF character = "\\" THEN
            char_width := 42;
        ELSEIF character = "^" THEN
            char_width := 38;
        ELSEIF character = "_" THEN
            char_width := 38;
        ELSEIF character = "`" THEN
            char_width := 18;
        ELSEIF character = "a" THEN
            char_width := 30;
        ELSEIF character = "b" THEN
            char_width := 30;
        ELSEIF character = "c" THEN
            char_width := 30;
        ELSEIF character = "d" THEN
            char_width := 30;
        ELSEIF character = "e" THEN
            char_width := 30;
        ELSEIF character = "f" THEN
            char_width := 22;
        ELSEIF character = "g" THEN
            char_width := 30;
        ELSEIF character = "h" THEN
            char_width := 28;
        ELSEIF character = "i" THEN
            char_width := 10;
        ELSEIF character = "j" THEN
            char_width := 18;
        ELSEIF character = "k" THEN
            char_width := 28;
        ELSEIF character = "l" THEN
            char_width := 6;
        ELSEIF character = "m" THEN
            char_width := 50;
        ELSEIF character = "n" THEN
            char_width := 28;
        ELSEIF character = "o" THEN
            char_width := 32;
        ELSEIF character = "p" THEN
            char_width := 30;
        ELSEIF character = "q" THEN
            char_width := 30;
        ELSEIF character = "r" THEN
            char_width := 22;
        ELSEIF character = "s" THEN
            char_width := 28;
        ELSEIF character = "t" THEN
            char_width := 22;
        ELSEIF character = "u" THEN
            char_width := 28;
        ELSEIF character = "v" THEN
            char_width := 30;
        ELSEIF character = "w" THEN
            char_width := 38;
        ELSEIF character = "x" THEN
            char_width := 28;
        ELSEIF character = "y" THEN
            char_width := 32;
        ELSEIF character = "z" THEN
            char_width := 28;
        ELSEIF character = "{" THEN
            char_width := 16;
        ELSEIF character = "}" THEN
            char_width := 16;
        ELSEIF character = "|" THEN
            char_width := 6;
        ELSEIF character = "~" THEN
            char_width := 42;
        ENDIF

        RETURN char_width;
    ENDFUNC

    !***********************************************************
    !
    ! Function get_word_width
    !   This function returns the written width of a given string
    !
    ! Example
    !   VAR string input_string := "hello";
    !   VAR num character_spacing := 2;
    !   VAR num word_width := get_word_width(input_string, character_spacing);
    !
    !***********************************************************
    FUNC num get_word_width(string word, num character_spacing)
        ! Define variables to be used later
        VAR num word_width := 0;
        VAR string character := "";
        VAR num string_length := 0;
        VAR num character_width := 0;

        ! Update string length
        string_length := StrLen(word);

        ! Calculate word width
        FOR index FROM 1 TO string_length DO
            character := StrPart(word, index, 1);
            character_width := get_character_width(character);

            word_width := word_width + character_width;
        ENDFOR

        ! Add character spacing
        word_width := word_width + (character_spacing * (string_length - 1.0));

        RETURN word_width;
    ENDFUNC

    !***********************************************************
    !
    ! Function get_ideal_font_size
    !   This function returns the ideal font size to ensure that a given string
    !   fits a particular view.
    !
    ! Example
    !   VAR string input_string := "hello, world";
    !   VAR num page_width := 250;
    !   VAR num padding := 10;
    !   VAR num font_size := get_ideal_font_size(input_string, page_width, padding);
    !
    !***********************************************************
    FUNC num get_ideal_font_size(string input_string, num page_width, num padding)
        ! Define max string length
        VAR num max_string_length := 20;

        ! Intialize a buffer to store the ideal word_length
        VAR num ideal_word_length := 0;

        ! Define variables to be used later
        VAR num ideal_font_size := 1.0;
        VAR num string_length := 0;
        VAR num word_length := 0;
        VAR num character_spacing := 2;

        string_length := StrLen(input_string);
        IF string_length > max_string_length THEN
            ! Truncate the input string if it exceeds the max allowed length
            input_string := StrPart(input_string, 0, max_string_length);
        ENDIF

        ! Update string length
        string_length := StrLen(input_string);

        ! Calculate word length
        word_length := get_word_width(input_string, character_spacing);

        ! Calculate ideal word length
        ideal_font_size := 1.0;
        ideal_word_length := page_width - (2.0 * padding);
        ideal_font_size := ideal_word_length / word_length;

        RETURN ideal_font_size;
    ENDFUNC

    !***********************************************************
    !
    ! Procedure DrawString
    !   This procedure draws a given string on the work surface
    !
    ! Example
    !   VAR string input_string := "Hello";    // String to write
    !   VAR num font_size := 1.0;              // Size of characters
    !   VAR speeddata approach_speed := v100;  // Approach speed for arm
    !   VAR speeddata write_speed := v80;      // Write speed for arm
    !   VAR num x_offset := 0;                 // x offset from worksurface origin
    !   VAR num y_offset := 0;                 // y offset from worksurface origin
    !   VAR num z_offset := 0;                 // z offset from worksurface origin
    !   VAR num pen_offset := 30;              // Defines pen position for pen up
    !
    !   DrawString input_string, font_size, approach_speed, write_speed, x_offset, y_offset, z_offset, penup_offset;
    !
    !***********************************************************
    PROC DrawString(string input_string, num font_size, speeddata approach_speed, speeddata write_speed, num x_offset, num y_offset, num z_offset, num penup_offset)
        ! Define default character size and input_string length
        VAR num char_width := 45;
        VAR num char_height := 50;
        VAR num input_length := 0;

        ! Define size of work surface
        VAR num page_width := 290;
        VAR num page_height := 400;

        ! Define start position
        VAR num start_x_offset := 0;
        VAR num start_y_offset := 0;
        VAR string character := "";

        ! Apply intial start offset
        start_x_offset := x_offset;
        start_y_offset := y_offset;

        ! Ensure that the font_size is not (zero | negative)
        IF font_size <= 0 THEN
            font_size := 0.1;
        ENDIF

        ! Update character height to based on font_size
        char_height := char_height * font_size;
        input_length := StrLen(input_string);

        ! Loop through the given input_string
        FOR index FROM 1 TO input_length DO
            ! Select the character at this index
            character := StrPart(input_string, index, 1);

            ! Draw the character
            DrawCharacter character, font_size, approach_speed, write_speed, x_offset, y_offset, z_offset, penup_offset;

            char_width := get_character_width(character);

            ! Update the width of the character based on font_size & move the arm #UpdateCursor
            char_width := (char_width + 2) * font_size;
            x_offset := x_offset + char_width;

            ! Engage text-wrap if arm at page width
            IF (x_offset + char_width) > page_width THEN
                x_offset := start_x_offset;
                y_offset := y_offset + char_height;
            ENDIF

            ! Engage page-wrap if arm at page-height
            IF (y_offset + char_height) > page_height THEN
                y_offset := start_y_offset;
                x_offset := start_x_offset;
            ENDIF
        ENDFOR

    ENDPROC

